// NETWORK 41
//   axisdata[4].Axis_Inbb: A-0-0021.13 -RD- Axis is ready for power to the amplifier (bb)
//   FP_C_0_0051: Operating hour counter
//   drive4: Real axis "Drive4" with axis number 4
//   r_operation_hour: FP_C_0_0051,Operation hour counter
fb_read_operation_hour(
    Enable := axisdata[4].Axis_Inbb,
    ParameterNumber := FP_C_0_0051,
    Axis := drive4,
    Value => r_operation_hour); // MB_ReadParameter

// NETWORK 42
//   axisdata[1].Axis_Inbb: A-0-0021.13 -RD- Axis is ready for power to the amplifier (bb)
//   FP_s_0_0189: Following distance
//   drive1: Real axis "Drive1" with axis number 1
//   r_following_11: FP_s_0_0189,following error
fb_read_s189_1(
    Enable := axisdata[1].Axis_Inbb,
    ParameterNumber := FP_s_0_0189,
    Axis := drive1,
    Value => r_following_11); // MB_ReadRealParameter

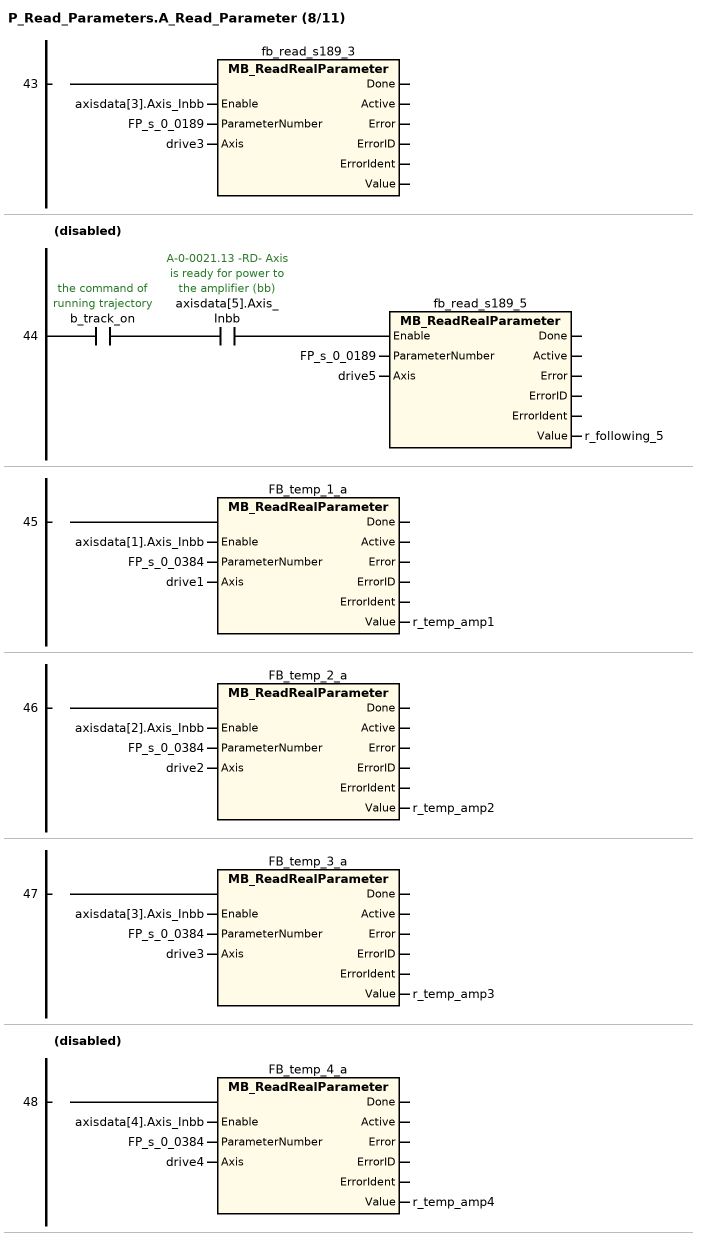
// NETWORK 43
//   axisdata[3].Axis_Inbb: A-0-0021.13 -RD- Axis is ready for power to the amplifier (bb)
//   FP_s_0_0189: Following distance
//   drive3: Real axis "Drive3" with axis number 3
fb_read_s189_3(Enable := axisdata[3].Axis_Inbb, ParameterNumber := FP_s_0_0189, Axis := drive3); // MB_ReadRealParameter

// NETWORK 44 (disabled)
//   b_track_on: the command of running trajectory
//   axisdata[5].Axis_Inbb: A-0-0021.13 -RD- Axis is ready for power to the amplifier (bb)
//   FP_s_0_0189: Following distance
//   drive5: Real axis "Drive5" with axis number 5
// fb_read_s189_5(
//     Enable := b_track_on AND axisdata[5].Axis_Inbb,
//     ParameterNumber := FP_s_0_0189,
//     Axis := drive5,
//     Value => r_following_5); // MB_ReadRealParameter

// NETWORK 45
//   axisdata[1].Axis_Inbb: A-0-0021.13 -RD- Axis is ready for power to the amplifier (bb)
//   FP_s_0_0384: Amplifier temperature
//   drive1: Real axis "Drive1" with axis number 1
//   r_temp_amp1: FP_S_0_0384,Amplifier temperature
FB_temp_1_a(
    Enable := axisdata[1].Axis_Inbb,
    ParameterNumber := FP_s_0_0384,
    Axis := drive1,
    Value => r_temp_amp1); // MB_ReadRealParameter

// NETWORK 46
//   axisdata[2].Axis_Inbb: A-0-0021.13 -RD- Axis is ready for power to the amplifier (bb)
//   FP_s_0_0384: Amplifier temperature
//   drive2: Real axis "Drive2" with axis number 2
FB_temp_2_a(
    Enable := axisdata[2].Axis_Inbb,
    ParameterNumber := FP_s_0_0384,
    Axis := drive2,
    Value => r_temp_amp2); // MB_ReadRealParameter

// NETWORK 47
//   axisdata[3].Axis_Inbb: A-0-0021.13 -RD- Axis is ready for power to the amplifier (bb)
//   FP_s_0_0384: Amplifier temperature
//   drive3: Real axis "Drive3" with axis number 3
FB_temp_3_a(
    Enable := axisdata[3].Axis_Inbb,
    ParameterNumber := FP_s_0_0384,
    Axis := drive3,
    Value => r_temp_amp3); // MB_ReadRealParameter

// NETWORK 48 (disabled)
//   axisdata[4].Axis_Inbb: A-0-0021.13 -RD- Axis is ready for power to the amplifier (bb)
//   FP_s_0_0384: Amplifier temperature
//   drive4: Real axis "Drive4" with axis number 4
// FB_temp_4_a(
//     Enable := axisdata[4].Axis_Inbb,
//     ParameterNumber := FP_s_0_0384,
//     Axis := drive4,
//     Value => r_temp_amp4); // MB_ReadRealParameter

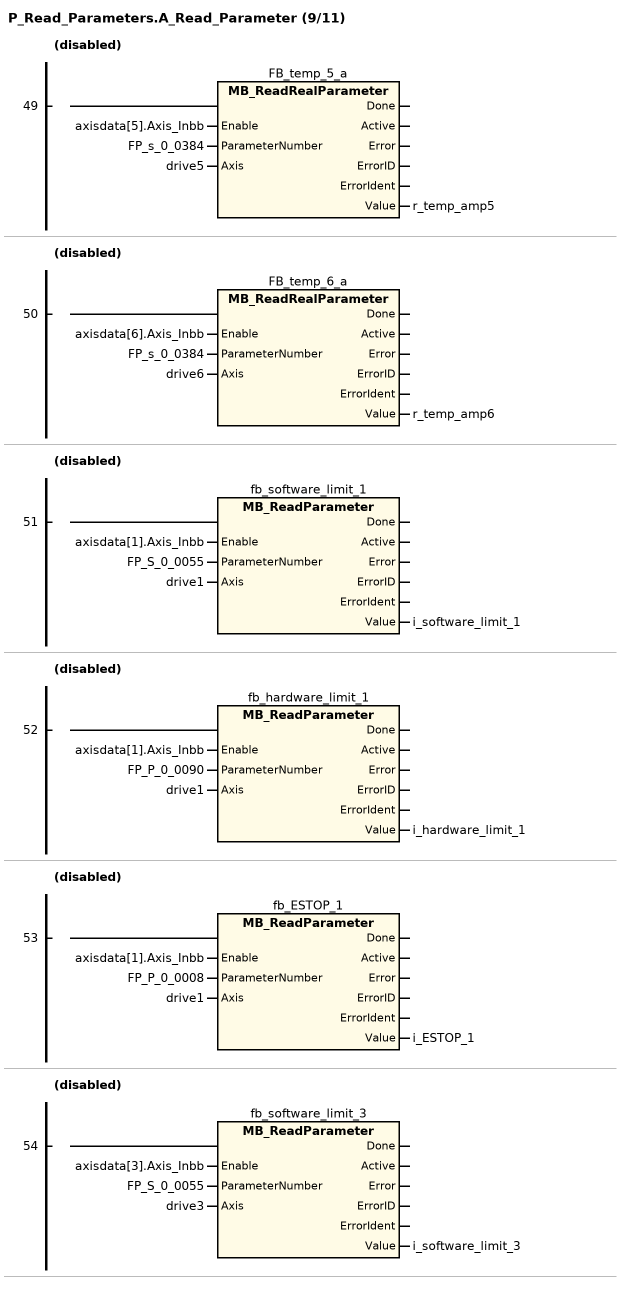
// NETWORK 49 (disabled)
//   axisdata[5].Axis_Inbb: A-0-0021.13 -RD- Axis is ready for power to the amplifier (bb)
//   FP_s_0_0384: Amplifier temperature
//   drive5: Real axis "Drive5" with axis number 5
// FB_temp_5_a(
//     Enable := axisdata[5].Axis_Inbb,
//     ParameterNumber := FP_s_0_0384,
//     Axis := drive5,
//     Value => r_temp_amp5); // MB_ReadRealParameter

// NETWORK 50 (disabled)
//   axisdata[6].Axis_Inbb: A-0-0021.13 -RD- Axis is ready for power to the amplifier (bb)
//   FP_s_0_0384: Amplifier temperature
//   drive6: Real axis "Drive6" with axis number 6
// FB_temp_6_a(
//     Enable := axisdata[6].Axis_Inbb,
//     ParameterNumber := FP_s_0_0384,
//     Axis := drive6,
//     Value => r_temp_amp6); // MB_ReadRealParameter

// NETWORK 51 (disabled)
//   fb_software_limit_1: test for limit check
//   axisdata[1].Axis_Inbb: A-0-0021.13 -RD- Axis is ready for power to the amplifier (bb)
//   FP_S_0_0055: Position polarities
//   drive1: Real axis "Drive1" with axis number 1
// fb_software_limit_1(
//     Enable := axisdata[1].Axis_Inbb,
//     ParameterNumber := FP_S_0_0055,
//     Axis := drive1,
//     Value => i_software_limit_1); // MB_ReadParameter

// NETWORK 52 (disabled)
//   axisdata[1].Axis_Inbb: A-0-0021.13 -RD- Axis is ready for power to the amplifier (bb)
//   FP_P_0_0090: Travel range limit parameter
//   drive1: Real axis "Drive1" with axis number 1
// fb_hardware_limit_1(
//     Enable := axisdata[1].Axis_Inbb,
//     ParameterNumber := FP_P_0_0090,
//     Axis := drive1,
//     Value => i_hardware_limit_1); // MB_ReadParameter

// NETWORK 53 (disabled)
//   axisdata[1].Axis_Inbb: A-0-0021.13 -RD- Axis is ready for power to the amplifier (bb)
//   FP_P_0_0008: Activation E-Stop function
//   drive1: Real axis "Drive1" with axis number 1
// fb_ESTOP_1(
//     Enable := axisdata[1].Axis_Inbb,
//     ParameterNumber := FP_P_0_0008,
//     Axis := drive1,
//     Value => i_ESTOP_1); // MB_ReadParameter

// NETWORK 54 (disabled)
//   axisdata[3].Axis_Inbb: A-0-0021.13 -RD- Axis is ready for power to the amplifier (bb)
//   FP_S_0_0055: Position polarities
//   drive3: Real axis "Drive3" with axis number 3
// fb_software_limit_3(
//     Enable := axisdata[3].Axis_Inbb,
//     ParameterNumber := FP_S_0_0055,
//     Axis := drive3,
//     Value => i_software_limit_3); // MB_ReadParameter

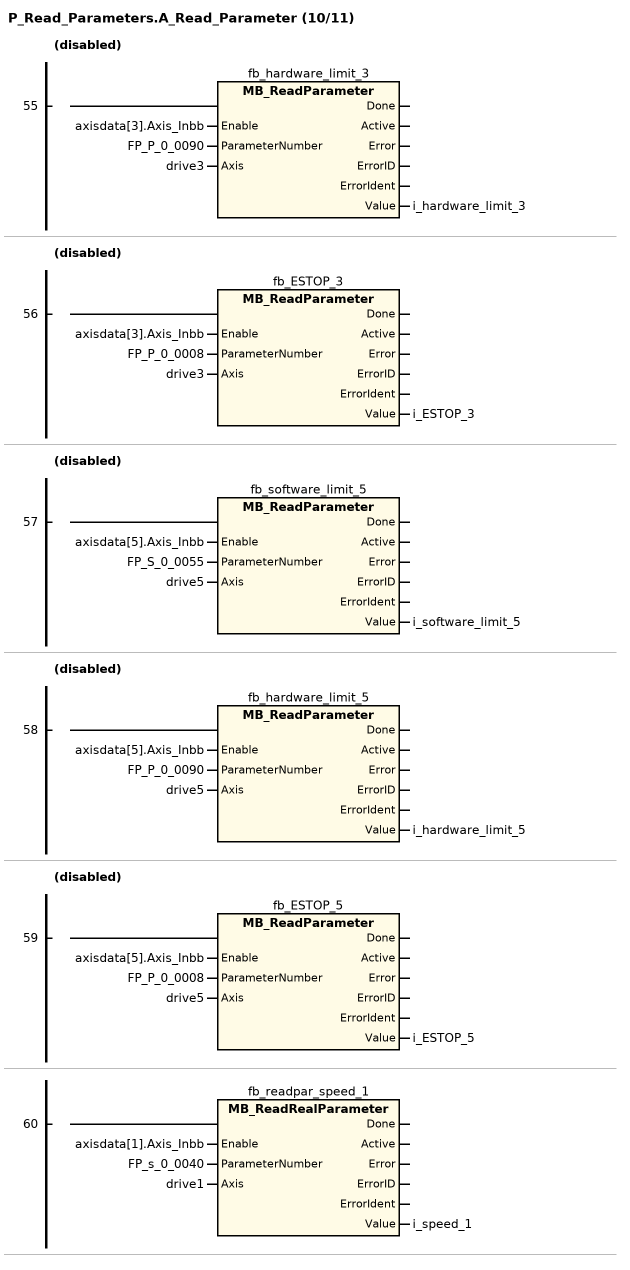
// NETWORK 55 (disabled)
//   axisdata[3].Axis_Inbb: A-0-0021.13 -RD- Axis is ready for power to the amplifier (bb)
//   FP_P_0_0090: Travel range limit parameter
//   drive3: Real axis "Drive3" with axis number 3
// fb_hardware_limit_3(
//     Enable := axisdata[3].Axis_Inbb,
//     ParameterNumber := FP_P_0_0090,
//     Axis := drive3,
//     Value => i_hardware_limit_3); // MB_ReadParameter

// NETWORK 56 (disabled)
//   axisdata[3].Axis_Inbb: A-0-0021.13 -RD- Axis is ready for power to the amplifier (bb)
//   FP_P_0_0008: Activation E-Stop function
//   drive3: Real axis "Drive3" with axis number 3
// fb_ESTOP_3(
//     Enable := axisdata[3].Axis_Inbb,
//     ParameterNumber := FP_P_0_0008,
//     Axis := drive3,
//     Value => i_ESTOP_3); // MB_ReadParameter

// NETWORK 57 (disabled)
//   axisdata[5].Axis_Inbb: A-0-0021.13 -RD- Axis is ready for power to the amplifier (bb)
//   FP_S_0_0055: Position polarities
//   drive5: Real axis "Drive5" with axis number 5
// fb_software_limit_5(
//     Enable := axisdata[5].Axis_Inbb,
//     ParameterNumber := FP_S_0_0055,
//     Axis := drive5,
//     Value => i_software_limit_5); // MB_ReadParameter

// NETWORK 58 (disabled)
//   axisdata[5].Axis_Inbb: A-0-0021.13 -RD- Axis is ready for power to the amplifier (bb)
//   FP_P_0_0090: Travel range limit parameter
//   drive5: Real axis "Drive5" with axis number 5
// fb_hardware_limit_5(
//     Enable := axisdata[5].Axis_Inbb,
//     ParameterNumber := FP_P_0_0090,
//     Axis := drive5,
//     Value => i_hardware_limit_5); // MB_ReadParameter

// NETWORK 59 (disabled)
//   axisdata[5].Axis_Inbb: A-0-0021.13 -RD- Axis is ready for power to the amplifier (bb)
//   FP_P_0_0008: Activation E-Stop function
//   drive5: Real axis "Drive5" with axis number 5
// fb_ESTOP_5(
//     Enable := axisdata[5].Axis_Inbb,
//     ParameterNumber := FP_P_0_0008,
//     Axis := drive5,
//     Value => i_ESTOP_5); // MB_ReadParameter

// NETWORK 60
//   axisdata[1].Axis_Inbb: A-0-0021.13 -RD- Axis is ready for power to the amplifier (bb)
//   FP_s_0_0040: Velocity feedback value
//   drive1: Real axis "Drive1" with axis number 1
//   i_speed_1: the velocity feedback value of motor1
fb_readpar_speed_1(
    Enable := axisdata[1].Axis_Inbb,
    ParameterNumber := FP_s_0_0040,
    Axis := drive1,
    Value => i_speed_1); // MB_ReadRealParameter

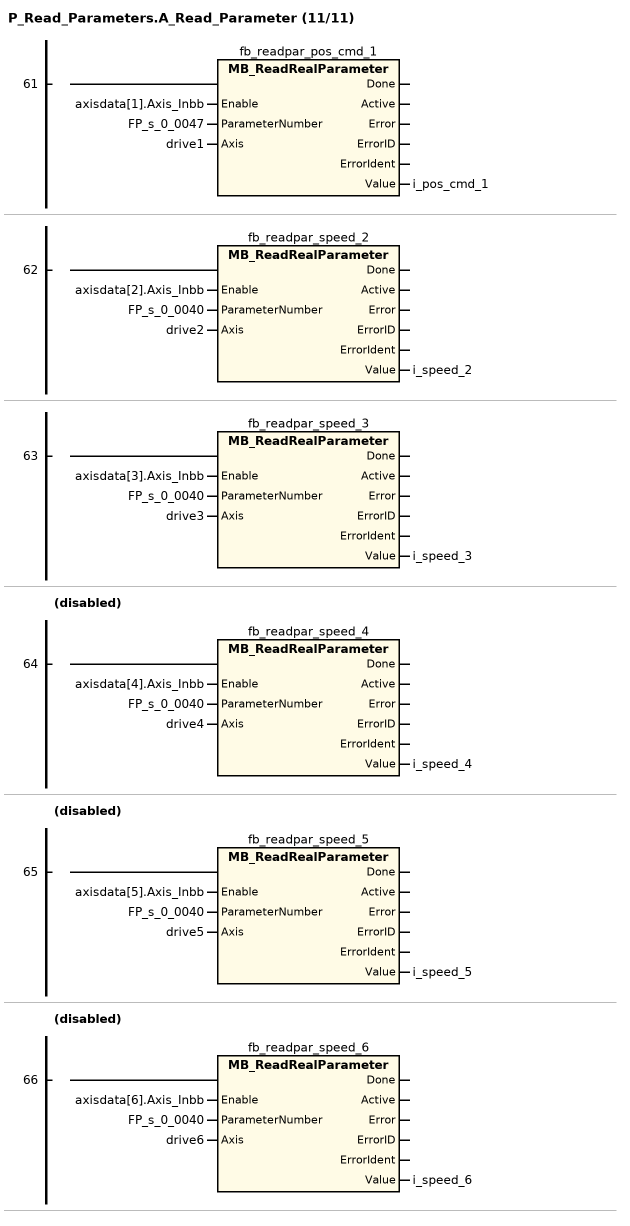
// NETWORK 61
//   axisdata[1].Axis_Inbb: A-0-0021.13 -RD- Axis is ready for power to the amplifier (bb)
//   FP_s_0_0047: Velocity feedback value
//   drive1: Real axis "Drive1" with axis number 1
//   i_pos_cmd_1: the velocity feedback value of motor1
fb_readpar_pos_cmd_1(
    Enable := axisdata[1].Axis_Inbb,
    ParameterNumber := FP_s_0_0047,
    Axis := drive1,
    Value => i_pos_cmd_1); // MB_ReadRealParameter

// NETWORK 62
//   axisdata[2].Axis_Inbb: A-0-0021.13 -RD- Axis is ready for power to the amplifier (bb)
//   FP_s_0_0040: Velocity feedback value
//   drive2: Real axis "Drive2" with axis number 2
//   i_speed_2: the velocity feedback value of motor1
fb_readpar_speed_2(
    Enable := axisdata[2].Axis_Inbb,
    ParameterNumber := FP_s_0_0040,
    Axis := drive2,
    Value => i_speed_2); // MB_ReadRealParameter

// NETWORK 63
//   axisdata[3].Axis_Inbb: A-0-0021.13 -RD- Axis is ready for power to the amplifier (bb)
//   FP_s_0_0040: Velocity feedback value
//   drive3: Real axis "Drive3" with axis number 3
//   i_speed_3: the velocity feedback value of motor3
fb_readpar_speed_3(
    Enable := axisdata[3].Axis_Inbb,
    ParameterNumber := FP_s_0_0040,
    Axis := drive3,
    Value => i_speed_3); // MB_ReadRealParameter

// NETWORK 64 (disabled)
//   axisdata[4].Axis_Inbb: A-0-0021.13 -RD- Axis is ready for power to the amplifier (bb)
//   FP_s_0_0040: Velocity feedback value
//   drive4: Real axis "Drive4" with axis number 4
//   i_speed_4: the velocity feedback value of motor1
// fb_readpar_speed_4(
//     Enable := axisdata[4].Axis_Inbb,
//     ParameterNumber := FP_s_0_0040,
//     Axis := drive4,
//     Value => i_speed_4); // MB_ReadRealParameter

// NETWORK 65 (disabled)
//   axisdata[5].Axis_Inbb: A-0-0021.13 -RD- Axis is ready for power to the amplifier (bb)
//   FP_s_0_0040: Velocity feedback value
//   drive5: Real axis "Drive5" with axis number 5
//   i_speed_5: the velocity feedback value of motor5
// fb_readpar_speed_5(
//     Enable := axisdata[5].Axis_Inbb,
//     ParameterNumber := FP_s_0_0040,
//     Axis := drive5,
//     Value => i_speed_5); // MB_ReadRealParameter

// NETWORK 66 (disabled)
//   axisdata[6].Axis_Inbb: A-0-0021.13 -RD- Axis is ready for power to the amplifier (bb)
//   FP_s_0_0040: Velocity feedback value
//   drive6: Real axis "Drive6" with axis number 6
//   i_speed_6: the velocity feedback value of motor1
// fb_readpar_speed_6(
//     Enable := axisdata[6].Axis_Inbb,
//     ParameterNumber := FP_s_0_0040,
//     Axis := drive6,
//     Value => i_speed_6); // MB_ReadRealParameter
END_ACTION

END_PROGRAM

// IndraMotionMlc1/Application/POUs/Motion/P_interpolator
(*This program is built for running trajectory,and the trajectory runs by the rule y=ax^2+bx+c.
In this PROGRAM,there are two kinds OF FUNCTION blocks,ML_WriteCyclicPosition AND ML_OpenCyclicPositionChannel.
They are used for give the position command value to the virtual axis.*)
PROGRAM P_interpolator
VAR
(*azimuth,elevation and FeedIndexer position at i_start point *)
	p1_az: LREAL;
	p1_el: LREAL;
	p1_FI: LREAL;
(*azimuth,elevation and FeedIndexer position at i_start+1 point*)
	p2_az: LREAL;
	p2_el: LREAL;
	p2_FI: LREAL;
(*azimuth,elevation and FeedIndexer position at i_start+2 point*)
	p3_az: LREAL;
	p3_el: LREAL;
	p3_FI: LREAL;
(*the facters of the formula y=ax^2+bx+c*)
	a_az: LREAL;
	b_az: LREAL;
	a_el: LREAL;
	b_el: LREAL;
	a_FI: LREAL;
	b_FI: LREAL;
	t: LREAL;
	t1: LREAL;(*the time at i_start point*)
	t2: LREAL;(*the time at i_start+1 point*)
	t3: LREAL;(*the time at i_start+2 point*)
	
(*<<<<<<<<<<<<<<<<<<<<<<<<Write a Position value to azimuth,elevation and FeedIndexer virtual axis>>>>>>>>>>>>>>>>>>*)
	fb_write_positon_az: ML_WriteCyclicPosition;
	fb_write_positon_el: ML_WriteCyclicPosition;
	fb_write_positon_FI: ML_WriteCyclicPosition;

(*Open Cyclic Position Channel for azimuth,elevation and FeedIndexer.
Only if the cyclic position target value channel is open, 
the position command will become effective in the next cycle on the axis.*)
	fb_open_channel_az: ML_OpenCyclicPositionChannel;
	fb_open_channel_el: ML_OpenCyclicPositionChannel;
	fb_open_channel_FI: ML_OpenCyclicPositionChannel;

(*<<<<<<<<<<<<<definition for rtrig>>>>>>>>>>>>>>*)
	rtrig_track_on: R_TRIG;
	rtrig_write_position: R_TRIG;
	rtrig_reset_open_channel: R_TRIG;
	rtrig_reset_goto_track: R_TRIG;
	r_rtrig_start_stop:R_TRIG;
	ton_track_on:TON;
	b_signal_for_open: BOOL;
(*<<<<<<<<<<<<<<<<<<<<<<<the current position>>>>>>>>>>>>>>>>>>>*)
	r_last_position_az: LREAL;
	r_last_position_el: LREAL;
	r_last_position_FI: LREAL;
(*<<<<<<<<<<<<<<<<<<<<<<<<<<the current speed>>>>>>>>>>>>>>>>>>>>*)
	r_vel_last_az: LREAL;
	r_vel_last_el: LREAL;
	r_vel_last_FI: LREAL;
(*the distance and time between the current point and the first point*)
	r_start_distance_az: LREAL;
	r_start_distance_el: LREAL;
	r_start_distance_FI: LREAL;
	r_time_distance: LREAL;
(*the current velocity *)
	r_vel_start_az: LREAL;
	r_vel_start_el: LREAL;
	r_vel_start_FI: LREAL;
(*the transition for the azimuth position,r_write_position_az.*)
	r_calc_pos_az:LREAL;
	V0_el: LREAL;
	V0_az: LREAL;
	V0_FI: LREAL;
	i_point_caught: INT:=1;
	V_start_az: LREAL;
	V_start_el: LREAL;
	V_start_FI: LREAL;
	i_caught_MJD1:LREAL;
	i_caught_MJD2:LREAL;
	i_caught_TAIoffset1:LREAL;
	i_caught_TAIoffset2:LREAL;
	b_test:BOOL;
	
	i_start_first:INT;
	i_end_first:INT;
	
	test_1:INT;
	test_2:INT;
	
	r_start_az:LREAL;
	r_caught_az:LREAL;
	
	ton_pause_on:TON;
	rtrig_pause_on:R_TRIG;
	r_abs_az_speed:LREAL; // units deg/sec
	r_abs_el_speed:LREAL; // units deg/sec
	test_enable_el: BOOL;
	b_start_to_compensate: BOOL;
	p_covert_velocity:LREAL;
	r_following_test: LREAL;
	r_following_31: LREAL;
	r_following_333: LREAL;
	p_covert_velocity_el: LREAL;	
	(**********offset************)
	r_az_offset_Vmax:LREAL:=2.0;
	r_el_offset_Vmax:LREAL:=0.85;
	r_az_offset_acc:LREAL:=1.0;
	r_el_offset_acc:LREAL:=0.25;
	r_az_offset_dec:LREAL:=0.5;
	r_el_offset_dec:LREAL:=0.25;
	r_old_offset_az:LREAL;
	r_old_offset_el:LREAL;
	r_new_offset_az:LREAL;
	r_new_offset_el:LREAL;

	r_test_offset_az_abs:LREAL;
	r_test_offset_el_abs:LREAL;
	i_test_offset_count:DINT:=0;
	r_offset_t1_acc:LREAL;
	r_offset_t2_v:LREAL;
	r_offset_t3_dec:LREAL;
	l_offset_t1_acc:LREAL;
	l_offset_t2_v:LREAL;
	l_offset_t3_dec:LREAL;
	r_offset_t1_acc_el:LREAL;
	r_offset_t2_v_el:LREAL;
	r_offset_t3_dec_el:LREAL;
	l_offset_t1_acc_el:LREAL;
	l_offset_t2_v_el:LREAL;
	l_offset_t3_dec_el:LREAL;
	r_offset_t:LREAL:=0;
	test_t:LREAL;
	r_az_offset_abs:LREAL;
	
	Static_done: BOOL;
	r_write_position_az_s: LREAL;
	r_write_position_el_s: LREAL;
	s_mp: StaticPmParam;
	Az_rad: LREAL;
	El_rad: LREAL;
	ABphi_rad: LREAL;
	TE: INT;
	//r_write_position_az_out: LREAL;
	//r_write_position_el_out: LREAL;
	test1: BOOL;
	Test2: BOOL;
	test3: BOOL;
	test4: BOOL;
	test5: BOOL;
	test6: BOOL;
	test7: BOOL;
	test8: BOOL;
	test9: BOOL;
	rtrig_write_position_sim: R_TRIG;
	fb_move_sim_track_Az: MC_MoveAbsolute;
	b_sim_trk_az_done: BOOL;
	b_sim_trk_el_done: BOOL;
	rtrig_reset_sim: R_TRIG;
	rtrig_reset_sim_move: R_TRIG;
	fb_move_sim_track_El: MC_MoveAbsolute;
	b_sim_write_az: BOOL;
	b_sim_trk_az_active: BOOL;
	TON_0: TON;
	b_sim_trk_el_active: BOOL;
	b_sim_trk_az_active_not: BOOL;
	f_trig_sim: F_TRIG;
	R_TRIG_0: R_TRIG;
	F_TRIG_0: F_TRIG;
	F_TRIG_1: F_TRIG;
	TON_1: TON;
	IL_EnableInOpBase_0: IL_SIGNALGENERATORTYPE01;
	TP_0: TP;
	TP_1: TP;
	TP_2: TP;
	BLINK_0: BLINK;
	b_sim_trk_exec: BOOL;
END_VAR

(*IF test_enable_el THEN
arAxisCtrl_gb[Drive3.AxisNo].Admin._OpMode.en := Modeah;
ELSE
arAxisCtrl_gb[Drive3.AxisNo].Admin._OpMode.en := Modeab;
END_IF
*)
//axisdata[3].dwUserCmdDataA_q.REAL_;

//axisdata[3].dwUserActualDataA_i.REAL_;



//axisdata[3].dwUserCmdDataA_q.REAL_:=axisdata[3].dwUserActualDataA_i.REAL_;





(*<<<<<<<<<<<<<<<<<<<<<calculate the current point in the stack>>>>>>>>>>>>>>>>>>>>>>>*)
//WHILE lr_MJD_current >= track_table[F_I_number(i_start+1)].MJD DO
test1:=lr_TAIoffset_current >= track_table[F_I_number(i_start+1)].TAIoffset;
WHILE lr_TAIoffset_current >= track_table[F_I_number(i_start+1)].TAIoffset DO
	IF i_start= i_end THEN
		EXIT;
	ELSE
		i_start:=F_I_number(i_start+1);
	END_IF;
END_WHILE


(*<<<<<<<<<<<<<<<<<<calculate the number of the points left in the stack>>>>>>>>>>>>>>*)
IF i_start=i_end THEN
	i_num_stack_left:=0;
ELSE
	i_num_stack_left:= i_end-i_start+1;
	IF i_num_stack_left<=0 THEN
		i_num_stack_left:=i_num_stack_left+i_total;
	END_IF;
END_IF

(* I Don't know what this piece of code is meant to do commenting it out 8/8/2024
IF i_num_stack_left>10 AND b_remote_on_run AND b_track_on=FALSE THEN
	b_track_on:=TRUE;
END_IF; *)


r_abs_az_speed:=ABS(AxisData[1].rActualVelocity_i)*6;
p_covert_velocity:=(0.5773*r_abs_az_speed*r_abs_az_speed*r_abs_az_speed - 0.4526*r_abs_az_speed*r_abs_az_speed + 11.313*r_abs_az_speed + 4.523)*0.2535;
p_covert_velocity_el:=0.5773*r_vel_EL*r_vel_EL*r_vel_EL - 0.4526*r_vel_EL*r_vel_EL + 11.313*r_vel_EL + 4.523;
(*<<<<<<<<<<<<<<<<<<<<<<<<<<<<<<<<<<<<<<the definication of trigger and TON>>>>>>>>>>>>>>>>>>>>>>>>>>>>>>>>>>>>>>>>>>>>>>>*)
r_rtrig_start_stop(clk:=b_track_on);(*before tracking ,stop the motion*)
ton_track_on(IN:=b_track_on,PT:=T#200MS);(*by using 200ms,program can search about 60 points*)
rtrig_track_on(clk:=ton_track_on.Q);(*the trigger for the initializtion*)


ton_pause_on(IN:=b_Track_Pause,PT:=T#4000MS);(*by using 200ms,program can search about 60 points*)
rtrig_pause_on(clk:=ton_pause_on.Q);(*the trigger for the initializtion*)

IF rtrig_pause_on.Q THEN
	b_track_on:=FALSE;
END_IF


(*<<<<<<<<<<<<<<<<<<<<<<<<<<<<main program of track>>>>>>>>>>>>>>>>>>>>>>>>>>>>>*)
IF b_track_on=TRUE THEN
	
(*<<<<<<<<<<<<<<<<<<<<<<<<<<< Calculate the tracking error>>>>>>>>>>>>>>>>>>>>>>>>>>>>>*)
	
	//IF ABS(track_table[i_start].MJD-lr_mjd_current)*86400<0.001 THEN
	Test2:=ABS(track_table[i_start].TAIoffset-lr_TAIoffset_current)<0.001;
	IF ABS(track_table[i_start].TAIoffset-lr_TAIoffset_current)<0.001 THEN
		r_following_1:=(r_pos_az_v-track_table[i_start].Azimuth);
		IF  ABS(r_following_1)<0.5  THEN
		   r_following_1:=(r_pos_az_v-track_table[i_start].Azimuth)/p_covert_velocity;
		END_IF
		   r_following_3:=(r_pos_el_v-track_table[i_start].Elevation);
		IF ABS(r_following_3)>0.0001 AND ABS(r_following_3)<=0.003 THEN
			r_following_3:=(r_pos_el_v-track_table[i_start].Elevation)/1.5;
		END_IF
		IF ABS(r_following_3)>0.003 AND ABS(r_following_3)<=0.006 THEN
			r_following_3:=(r_pos_el_v-track_table[i_start].Elevation)/2;
		END_IF
		IF ABS(r_following_3)>0.006 AND ABS(r_following_3)<=0.02 THEN
			r_following_3:=(r_pos_el_v-track_table[i_start].Elevation)/4;
		END_IF
		r_following_radius_asec := LREAL_TO_REAL((SQRT(EXPT(r_following_1,2)+EXPT(r_following_3,2)))*3600);  // Following erroring terms of a radius. 
	END_IF
(*
	IF ABS(r_following_3)> ABS(r_track_error[2]) THEN	
		r_following_33:=r_track_error[2];
	ELSE
		r_following_33:=r_following_33;
	END_IF
		IF ABS(r_following_33)>0.01 THEN
			r_following_33:=r_following_33/10;
		END_IF
	IF ABS(r_vel_EL)<0.0001 THEN
		r_following_3:=r_following_33;
	ELSE
		r_following_3:=r_following_33/p_covert_velocity_el;
	END_IF	
*)	
(*<<<<<<<<<<<<when finish all the points or the power is down,then reset the track_on>>>>>>>>>>>>>>>>>>>*)
	IF i_start=i_end OR b_remote_on_run=FALSE THEN
		 b_track_on:=FALSE;
	END_IF
(*<<<<<<<<<<<<<<<<<<<<<<<<<<<<stop the motion before tracking>>>>>>>>>>>>>>>>>>>*)
	IF r_rtrig_start_stop.Q THEN
		b_SCC_STOP:=TRUE;
	END_IF
	IF rtrig_track_on.Q=TRUE THEN
(*<<<<<<<<<<<<<<<<<<<<<<<<<<<<<<find the first point which can be caught up>>>>>>>>>>>>>>>>>>>>>>>>>>>*)
		//WHILE ABS(track_table[i_start].Azimuth-r_pos_az_v)/((track_table[i_start].MJD-lr_mjd_current)*86400-0.05)>2.9 OR (track_table[i_start].MJD-lr_mjd_current)*86400-0.05<0 DO
		test3:=ABS(track_table[i_start].Azimuth-r_pos_az_v)/((track_table[i_start].TAIoffset-lr_TAIoffset_current)-0.05)>2.9 OR (track_table[i_start].TAIoffset-lr_TAIoffset_current)-0.05<0;
		WHILE ABS(track_table[i_start].Azimuth-r_pos_az_v)/((track_table[i_start].TAIoffset-lr_TAIoffset_current)-0.05)>2.9 OR (track_table[i_start].TAIoffset-lr_TAIoffset_current)-0.05<0 DO
		//WHILE ABS(entry_buffer1[i_start].Azimuth-r_pos_az_v)/((entry_buffer1[i_start].MJD-lr_mjd_current)*86400-0.05)>2.9 DO
			IF i_start=i_end-3 THEN
				EXIT;
			ELSE
				i_start:=F_I_number(i_start+1);
			END_IF
		END_WHILE
		
		//WHILE ABS(track_table[i_start].Elevation-r_pos_el)/((track_table[i_start].MJD-lr_mjd_current)*86400-0.05)>0.8 OR (track_table[i_start].MJD-lr_mjd_current)*86400-0.05<0 DO
		test4:=ABS(track_table[i_start].Elevation-r_pos_el)/((track_table[i_start].TAIoffset-lr_TAIoffset_current)-0.05)>0.8 OR (track_table[i_start].TAIoffset-lr_TAIoffset_current)-0.05<0;
		WHILE ABS(track_table[i_start].Elevation-r_pos_el)/((track_table[i_start].TAIoffset-lr_TAIoffset_current)-0.05)>0.8 OR (track_table[i_start].TAIoffset-lr_TAIoffset_current)-0.05<0 DO	
		//WHILE ABS(entry_buffer1[i_start].Elevation-r_pos_motor3)/((entry_buffer1[i_start].MJD-lr_mjd_current)*86400-0.05)>1000 DO
			IF i_start=i_end-3 THEN
				EXIT;
			ELSE
				i_start:=F_I_number(i_start+1);
			END_IF
		END_WHILE
(*		WHILE ABS(entry_buffer1[i_start].FeedIndexer-r_pos_FI_v)/((entry_buffer1[i_start].MJD-lr_mjd_current)*86400-0.05)>2 OR (entry_buffer1[i_start].MJD-lr_mjd_current)*86400-0.05<0 DO
			IF i_start=i_end-3 THEN
				EXIT;
			ELSE
				i_start:=F_I_number(i_start+1);
			END_IF
		END_WHILE
*)

//		arAxisCtrl_gb[Drive3.AxisNo].Admin._OpMode.en := ModeCyclicVelocity; 
		b_write_el_vel:=TRUE;
		i_point_caught:=i_start;
		//i_caught_MJD1:=track_table[i_point_caught].MJD;
		 i_caught_TAIoffset1:=track_table[i_point_caught].TAIoffset;
		//i_caught_MJD2:=lr_MJD_current;
		i_caught_TAIoffset2:=lr_TAIoffset_current;
		r_start_az:=r_pos_az_v;
		r_caught_az:=track_table[i_point_caught].Azimuth;
		
(*if the first point which can be caught up is the last one£¬reset track_on*)
		IF i_start=i_end-3 THEN
			b_track_on:=FALSE;
		ELSE
			//track_table[F_I_number(i_start-1)].MJD:=lr_MJD_current+0.0000008;(*(69ms)after gunner change p41 from 0 to 100ms*)
			track_table[F_I_number(i_start-1)].TAIoffset:=lr_TAIoffset_current+0.069;(*(69ms)after gunner change p41 from 0 to 100ms*)
			track_table[F_I_number(i_start-1)].Azimuth:=r_pos_az_v;
			track_table[F_I_number(i_start-1)].elevation:=r_pos_el;
(*			entry_buffer1[F_I_number(i_start-1)].FeedIndexer:=r_pos_FI_v;  *)
		i_start:=F_I_number(i_start-1);
		r_write_position_az:=track_table[i_start].Azimuth;
		r_write_position_el:=track_table[i_start].Elevation;
(*		r_write_position_FI:=entry_buffer1[i_start].FeedIndexer;   *)
		r_last_position_az:=r_write_position_az;
		r_last_position_el:=r_write_position_el;
(*		r_last_position_FI:=r_write_position_FI;   *)
		b_signal_for_open:=TRUE;
		END_IF

	END_IF
(*when the position is all nearby the start point,open the channel for writing position to all axis*)
test5:=b_signal_for_open AND (ABS(r_pos_az_v-track_table[i_start].Azimuth)<0.001) AND (ABS(r_pos_el-track_table[i_start].Elevation)<0.001);
	IF b_signal_for_open AND (ABS(r_pos_az_v-track_table[i_start].Azimuth)<0.001) AND (ABS(r_pos_el-track_table[i_start].Elevation)<0.001) THEN
		b_open_channel_az:=TRUE;
//		b_start_cyclicvel:=TRUE;
//		b_open_channel_el:=TRUE;
(*		b_open_channel_FI:=TRUE;*)
		b_signal_for_open:=FALSE;
	END_IF
(*defind the variables for calculating the cubic fuction*)
		//t:=lr_MJD_current;
		//t1:=track_table[i_start].MJD;
		//t2:=track_table[F_I_number(i_start+1)].MJD;
		//t3:=track_table[F_I_number(i_start+2)].MJD;
		t:=lr_TAIoffset_current;
		t1:=track_table[i_start].TAIoffset;
		t2:=track_table[F_I_number(i_start+1)].TAIoffset;
		t3:=track_table[F_I_number(i_start+2)].TAIoffset;
		p1_az:=track_table[i_start].Azimuth;
		p2_az:=track_table[F_I_number(i_start+1)].Azimuth;
		p3_az:=track_table[F_I_number(i_start+2)].Azimuth;
		
		r_test1:=p1_az;
		r_test2:=p2_az;
		r_test3:=p3_az;
		
		p1_el:=track_table[i_start].elevation;
		p2_el:=track_table[F_I_number(i_start+1)].elevation;
		p3_el:=track_table[F_I_number(i_start+2)].elevation;		
(*		p1_FI:=entry_buffer1[i_start].FeedIndexer;
		p2_FI:=entry_buffer1[F_I_number(i_start+1)].FeedIndexer;
		p3_FI:=entry_buffer1[F_I_number(i_start+2)].FeedIndexer;
*)		
		//i_start;
		test_1:=F_I_number(i_start+1);
		test_2:=F_I_number(i_start+2);
(*construct the first cubic section by 2 points and 2 velocity*)
(*	IF	lr_MJD_current<entry_buffer1[i_point_caught].MJD AND lr_MJD_current>entry_buffer1[F_I_number(i_point_caught-1)].MJD THEN  *)
	//IF	lr_MJD_current<i_caught_MJD1 AND lr_MJD_current>i_caught_MJD2 THEN
test6:=lr_TAIoffset_current<i_caught_TAIoffset1 AND lr_TAIoffset_current>i_caught_TAIoffset2;
 IF	lr_TAIoffset_current<i_caught_TAIoffset1 AND lr_TAIoffset_current>i_caught_TAIoffset2 THEN	
	
		IF b_track_on THEN
			V_start_az:=(p3_az-p2_az)/(t3-t2);
			V_start_el:=(p3_el-p2_el)/(t3-t2);
(*			V_start_FI:=(p3_FI-p2_FI)/(t3-t2);  *)
			v0_az:=V_start_az;
			v0_el:=V_start_el;
(*			v0_FI:=V_start_FI;   *)
			b_test:=TRUE;
			b_start_to_compensate:=TRUE;

			a_az:=V_start_az/(t2-t1)/(t2-t1)-2*(p2_az-p1_az)/(t2-t1)/(t2-t1)/(t2-t1);
			b_az:=3*(p2_az-p1_az)/(t2-t1)/(t2-t1)-V_start_az/(t2-t1);
			a_el:=V_start_el/(t2-t1)/(t2-t1)-2*(p2_el-p1_el)/(t2-t1)/(t2-t1)/(t2-t1);
			b_el:=3*(p2_el-p1_el)/(t2-t1)/(t2-t1)-V_start_el/(t2-t1);
(*			a_FI:=V_start_FI/(t2-t1)/(t2-t1)-2*(p2_FI-p1_FI)/(t2-t1)/(t2-t1)/(t2-t1);
			b_FI:=3*(p2_FI-p1_FI)/(t2-t1)/(t2-t1)-V_start_FI/(t2-t1);
*)
			r_write_position_az:=a_az*(t-t1)*(t-t1)*(t-t1)+b_az*(t-t1)*(t-t1)+p1_az;
			r_write_position_el:=a_el*(t-t1)*(t-t1)*(t-t1)+b_el*(t-t1)*(t-t1)+p1_el;
(*			r_write_position_FI:=a_FI*(t-t1)*(t-t1)*(t-t1)+b_FI*(t-t1)*(t-t1)+p1_FI;   *)
		END_IF
	ELSE
		IF i_num_stack_left>2 THEN
			IF b_track_on THEN
(*<<<<<<<<<<<<<<<<<<<<<<<<<<<<<calculate the a and b in the function y=ax^3+bx^2+cx+d>>>>>>>>>>>>>>>>>>>>>>*)
(*y=a*(x-x1)^3+b*(x-x1)^2+c(x-x1)+d,   c=v0,  d=y1*)
			a_az:=((p3_az-p1_az)/(t3-t1)/(t3-t1)-(p2_az-p1_az)/(t2-t1)/(t2-t1)-v0_az/(t3-t1)+v0_az/(t2-t1))/(t3-t2);
			b_az:=((p3_az-p1_az)*(t2-t1)/(t3-t1)/(t3-t1)-(p2_az-p1_az)*(t3-t1)/(t2-t1)/(t2-t1)-v0_az*(t2-t1)/(t3-t1)+v0_az*(t3-t1)/(t2-t1))/(t2-t3);
			a_el:=((p3_el-p1_el)/(t3-t1)/(t3-t1)-(p2_el-p1_el)/(t2-t1)/(t2-t1)-v0_el/(t3-t1)+v0_el/(t2-t1))/(t3-t2);
			b_el:=((p3_el-p1_el)*(t2-t1)/(t3-t1)/(t3-t1)-(p2_el-p1_el)*(t3-t1)/(t2-t1)/(t2-t1)-v0_el*(t2-t1)/(t3-t1)+v0_el*(t3-t1)/(t2-t1))/(t2-t3);
(*			a_FI:=((p3_FI-p1_FI)/(t3-t1)/(t3-t1)-(p2_FI-p1_FI)/(t2-t1)/(t2-t1)-v0_FI/(t3-t1)+v0_FI/(t2-t1))/(t3-t2);
			b_FI:=((p3_FI-p1_FI)*(t2-t1)/(t3-t1)/(t3-t1)-(p2_FI-p1_FI)*(t3-t1)/(t2-t1)/(t2-t1)-v0_FI*(t2-t1)/(t3-t1)+v0_FI*(t3-t1)/(t2-t1))/(t2-t3);
*)
b_test:=FALSE;
			//IF lr_MJD_current>=track_table[i_start].MJD AND lr_MJD_current<=track_table[F_I_number(i_start+1)].MJD THEN
			test7:=lr_TAIoffset_current>=track_table[i_start].TAIoffset AND lr_TAIoffset_current<=track_table[F_I_number(i_start+1)].TAIoffset;
			IF lr_TAIoffset_current>=track_table[i_start].TAIoffset AND lr_TAIoffset_current<=track_table[F_I_number(i_start+1)].TAIoffset THEN
			
				r_write_position_az:=a_az*(t-t1)*(t-t1)*(t-t1)+b_az*(t-t1)*(t-t1)+v0_az*(t-t1)+p1_az;
				r_write_position_el:=a_el*(t-t1)*(t-t1)*(t-t1)+b_el*(t-t1)*(t-t1)+v0_el*(t-t1)+p1_el;
				r_cyclic_velocity_test:=(p2_el-p1_el)/(t2-t1)/86400;
				//r_cyclic_velocity_test:=(p2_el-p1_el)/(t2-t1);
				r_cyclic_velocity:=V0_el/86400;
				// r_cyclic_velocity:=V0_el;
(*				r_write_position_FI:=a_FI*(t-t1)*(t-t1)*(t-t1)+b_FI*(t-t1)*(t-t1)+v0_FI*(t-t1)+p1_FI;   *)
			END_IF
(*calculate the velocity of the last point*)
			//IF (lr_MJD_current-track_table[F_I_number(i_start+1)].MJD)*86400>=-0.002 AND (lr_MJD_current-track_table[F_I_number(i_start+1)].MJD)*86400<0 THEN
			test8:=(lr_TAIoffset_current-track_table[F_I_number(i_start+1)].TAIoffset)>=-0.002 AND (lr_TAIoffset_current-track_table[F_I_number(i_start+1)].TAIoffset)<0;
			IF (lr_TAIoffset_current-track_table[F_I_number(i_start+1)].TAIoffset)>=-0.002 AND (lr_TAIoffset_current-track_table[F_I_number(i_start+1)].TAIoffset)<0 THEN
				V0_az:=3*a_az*(t2-t1)*(t2-t1)+2*b_az*(t2-t1)+v0_az;
				V0_el:=3*a_el*(t2-t1)*(t2-t1)+2*b_el*(t2-t1)+v0_el;
(*				V0_FI:=3*a_FI*(t2-t1)*(t2-t1)+2*b_FI*(t2-t1)+v0_FI;    *)
			END_IF
			END_IF
		ELSE
(*<<<<<<<<<<<<<<<<<<<<<<<<run the last two points>>>>>>>>>>>>>>>>>>>>>>>>>>*)
			IF b_track_on THEN 
				//IF lr_MJD_current>=track_table[i_start].MJD AND lr_MJD_current<=track_table[F_I_number(i_start+1)].MJD THEN
				test9:= lr_TAIoffset_current>=track_table[i_start].TAIoffset AND lr_TAIoffset_current<=track_table[F_I_number(i_start+1)].TAIoffset;
				IF lr_TAIoffset_current>=track_table[i_start].TAIoffset AND lr_TAIoffset_current<=track_table[F_I_number(i_start+1)].TAIoffset THEN
				r_write_position_az:=(p2_az-p1_az)*(t-t1)/(t2-t1)+p1_az;
				r_write_position_el:=(p2_el-p1_el)*(t-t1)/(t2-t1)+p1_el;
(*				r_write_position_FI:=((p2_FI-p1_FI)*(t-t1)/(t2-t1)+p1_FI);     *)
				END_IF
			END_IF
		END_IF
	END_IF

	
IF b_start_to_compensate THEN
//	r_offset_el:=r_compensation_value_motor;
	r_write_position_az:=r_write_position_az+r_test_offset_az;
	r_write_position_el:=r_write_position_el+r_test_offset_el;
//	r_write_position_el:=r_write_position_el+r_offset_el;
END_IF
	
(*<<<<<<<<<<<<<<<<<<<<<<<<<limit the trajectory speed >>>>>>>>>>>>>>>>>>>>>>>>>*)
(*Because the program runs every 2ms,so wo can limit the position by the rule ¦¤y<v*¦¤t.*)
(*Azimuth trajectory speed limit is 5.1¡ã/s*)


		IF r_write_position_az-r_last_position_az>0.0031 THEN
				r_write_position_az:=r_last_position_az+0.0031;
				b_track_overspeed_az:=1;
			ELSIF r_write_position_az-r_last_position_az<-0.0031 THEN
				r_write_position_az:=r_last_position_az-0.0031;
				b_track_overspeed_az:=1;
			ELSE
				b_track_overspeed_az:=0;
			END_IF
(*Elevation trajectory speed limit is 1.05¡ã/s*)
			IF r_write_position_el-r_last_position_el>0.00091 THEN
				r_write_position_el:=r_last_position_el+0.00091;
				b_track_overspeed_el:=1;
			ELSIF r_write_position_el-r_last_position_el<-0.00091 THEN
				r_write_position_el:=r_last_position_el-0.00091;
				b_track_overspeed_el:=1;
			ELSE
				b_track_overspeed_el:=0;
			END_IF
(*
(*FeedIndexer trajectory speed limit is 2.1¡ã/s*)
			IF r_write_position_FI-r_last_position_FI>0.0042 THEN
				r_write_position_FI:=r_last_position_FI+0.0042;
				b_track_overspeed_FI:=1;
			ELSIF r_write_position_FI-r_last_position_FI<-0.0042 THEN
				r_write_position_FI:=r_last_position_FI-0.0042;
				b_track_overspeed_FI:=1;
			ELSE
				b_track_overspeed_FI:=0;
			END_IF
*)
			
			
(*register the velocity and position for calculate the speed limit and acceleration limit*)
			r_last_position_az:=r_write_position_az;
			r_last_position_el:=r_write_position_el;
(*			r_last_position_FI:=r_write_position_FI;   *)
(*<<<<<<<<<<<<<<<<<<<<<<<<close the cyclic channel and reset the track error>>>>>>>>>>>>>>>>>>>>>>>>>>*)
ELSE
(*close the cyclic channel*)
	b_open_channel_az:=FALSE;
	b_open_channel_el:=FALSE;
	b_start_to_compensate:=FALSE;
	r_compensation_value_motor:=0;
(*	b_open_channel_FI:=FALSE;  *)
(*reset the following error and so on*)
    r_write_position_el:= axisdata[8].rActualPosition_i;
	r_write_position_az:=  axisdata[7].rActualPosition_i;
	r_track_error[1]:=0;
	r_track_error[2]:=0;
	r_track_error[3]:=0;
	V0_az:=0;
	V0_el:=0;
	V_start_az:=0;
	V_start_el:=0;
	IF NOT(b_SCC_goto) AND NOT(b_track_on) THEN 
		r_following_1:=0.00;
		r_following_3:=0.00;
	END_IF
END_IF

 IF  b_test_offset_start THEN
	 	r_offset_t:=r_offset_t+0.001;
		test_t:=r_offset_t-r_offset_t1_acc-r_offset_t2_v;
 		(*****************AZ offset**********)
		r_az_offset_abs:=ABS(r_offset_az);
		r_offset_t1_acc:=r_az_offset_Vmax/r_az_offset_acc;
	 	r_offset_t3_dec:=r_az_offset_Vmax/r_az_offset_dec;
	 	l_offset_t1_acc:=0.5*r_az_offset_acc*r_offset_t1_acc*r_offset_t1_acc;
	 	l_offset_t3_dec:=0.5*r_az_offset_dec*r_offset_t3_dec*r_offset_t3_dec;
 		r_offset_t2_v:=(r_az_offset_abs-l_offset_t1_acc-l_offset_t3_dec)/r_az_offset_Vmax;
		l_offset_t2_v:=r_az_offset_Vmax*r_offset_t2_v;

			IF r_offset_t <=r_offset_t1_acc THEN
				r_test_offset_az_abs:=0.5*r_az_offset_acc*r_offset_t*r_offset_t;
			ELSIF r_offset_t1_acc<r_offset_t AND r_offset_t<(r_offset_t1_acc+r_offset_t2_v) THEN 
				r_test_offset_az_abs:=r_test_offset_az_abs+0.001*r_az_offset_Vmax;
			ELSIF (r_offset_t1_acc+r_offset_t2_v)<=r_offset_t AND r_offset_t<(r_offset_t1_acc+r_offset_t2_v+r_offset_t3_dec) THEN
				r_test_offset_az_abs:=l_offset_t1_acc+l_offset_t2_v+(r_offset_t-r_offset_t1_acc-r_offset_t2_v)*r_az_offset_Vmax-0.5*r_az_offset_dec*(r_offset_t-r_offset_t1_acc-r_offset_t2_v)*(r_offset_t-r_offset_t1_acc-r_offset_t2_v);
			ELSE 
				r_test_offset_az_abs:=r_az_offset_abs;
			END_IF

		IF r_test_offset_az_abs>=r_az_offset_abs THEN
			r_test_offset_az_abs:=r_az_offset_abs;
		END_IF
		IF r_offset_az<0 THEN
			r_test_offset_az:=-r_test_offset_az_abs;
		ELSE 
			r_test_offset_az:=r_test_offset_az_abs;
		END_IF
		r_test_offset_az:=r_offset_az_old+r_test_offset_az;
		
		
			(*****************EL offset**********)
		r_el_offset_abs:=ABS(r_offset_el);
		r_offset_t1_acc_el:=r_el_offset_Vmax/r_el_offset_acc;
	 	r_offset_t3_dec_el:=r_el_offset_Vmax/r_el_offset_dec;
	 	l_offset_t1_acc_el:=0.5*r_el_offset_acc*r_offset_t1_acc_el*r_offset_t1_acc_el;
	 	l_offset_t3_dec_el:=0.5*r_el_offset_dec*r_offset_t3_dec_el*r_offset_t3_dec_el;
 		r_offset_t2_v_el:=(r_el_offset_abs-l_offset_t1_acc_el-l_offset_t3_dec_el)/r_el_offset_Vmax;
		l_offset_t2_v_el:=r_el_offset_Vmax*r_offset_t2_v_el;

			IF r_offset_t <=r_offset_t1_acc_el THEN
				r_test_offset_el_abs:=0.5*r_el_offset_acc*r_offset_t*r_offset_t;
			ELSIF r_offset_t1_acc_el<r_offset_t AND r_offset_t<(r_offset_t1_acc_el+r_offset_t2_v_el) THEN 
				r_test_offset_el_abs:=r_test_offset_el_abs+0.001*r_el_offset_Vmax;
			ELSIF (r_offset_t1_acc_el+r_offset_t2_v_el)<=r_offset_t AND r_offset_t<(r_offset_t1_acc_el+r_offset_t2_v_el+r_offset_t3_dec_el) THEN
				r_test_offset_el_abs:=l_offset_t1_acc_el+l_offset_t2_v_el+(r_offset_t-r_offset_t1_acc_el-r_offset_t2_v_el)*r_el_offset_Vmax-0.5*r_el_offset_dec*(r_offset_t-r_offset_t1_acc_el-r_offset_t2_v_el)*(r_offset_t-r_offset_t1_acc_el-r_offset_t2_v_el);
			ELSE 
				r_test_offset_el_abs:=r_el_offset_abs;
			END_IF

		IF r_test_offset_el_abs>=r_el_offset_abs THEN
			r_test_offset_el_abs:=r_el_offset_abs;
		END_IF
		IF r_offset_el<0 THEN
			r_test_offset_el:=-r_test_offset_el_abs;
		ELSE 
			r_test_offset_el:=r_test_offset_el_abs;
		END_IF
		r_test_offset_el:=r_offset_el_old+r_test_offset_el;
    IF 	r_test_offset_el_abs=r_el_offset_abs AND r_test_offset_az_abs=r_az_offset_abs THEN 	
		b_test_offset_start:=FALSE;
		b_offset_running:=FALSE;
	END_IF
				
ELSE
	i_test_offset_count:=0;
	r_offset_t:=0;
	r_offset_az_old:=r_test_offset_az;
	r_offset_el_old:=r_test_offset_el;
END_IF


P_Track_cubic.A_StaticPM();
P_Track_cubic.A_AmbTempPM();
P_Track_cubic.A_DynamicPM();


Tracking.Status.p_desired_El:=r_write_position_el-Tracking.Status.act_statOffset_value_El/gc_lr_arcsec2deg;
Tracking.Status.p_desired_Az:=r_write_position_az-(Tracking.Status.act_statOffset_value_Xel/gc_lr_arcsec2deg)/COS(ML_degtorad(r_write_position_el));

IF b_track_on THEN 
r_write_position_az_out:=r_write_position_az-Pointing.Status.StaticPmCorrVal_Az/gc_lr_arcsec2deg-Pointing.Status.TiltCorrVal_Az/gc_lr_arcsec2deg-Pointing.Status.AmbTempCorrVal_Az/gc_lr_arcsec2deg;
r_write_position_el_out:=r_write_position_el-Pointing.Status.StaticPmCorrVal_El/gc_lr_arcsec2deg-Pointing.Status.TiltCorrVal_El/gc_lr_arcsec2deg-Pointing.Status.AmbTempCorrVal_El/gc_lr_arcsec2deg;
END_IF

IF gc_b_sim_on THEN 
	P_Track_cubic.A_Sim_track_function_blocks();
ELSE	
	P_Track_cubic.A_track_fuction_blocks();
END_IF

ACTION A_track_fuction_blocks:
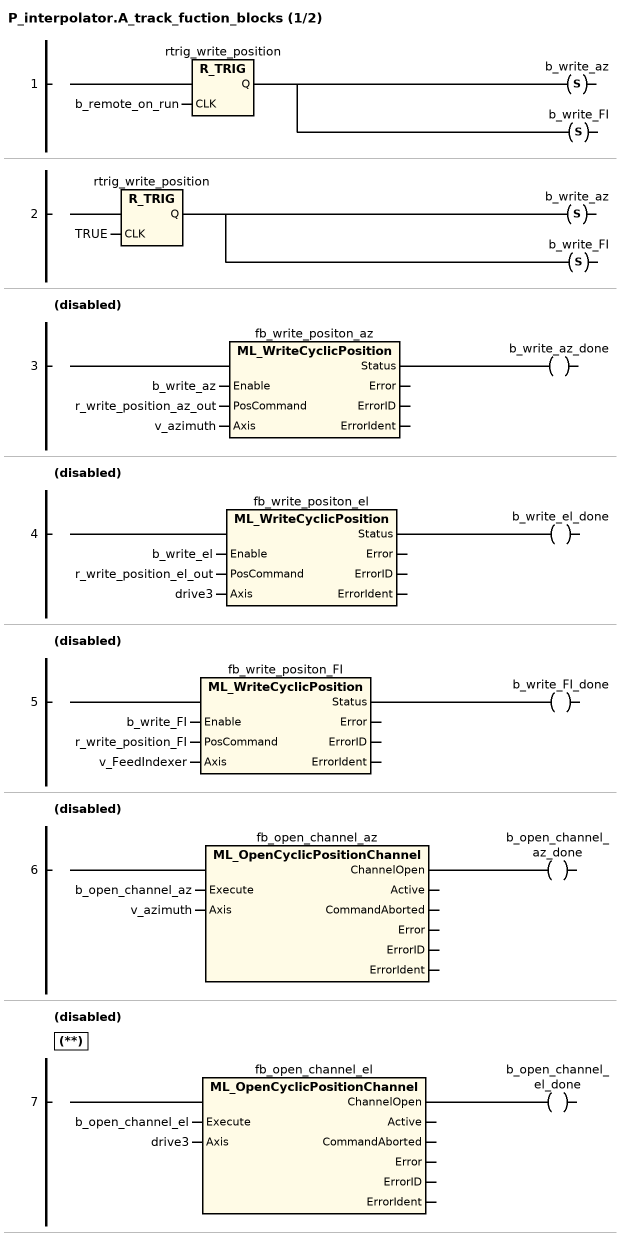
// NETWORK 1
rtrig_write_position(CLK := b_remote_on_run); // R_TRIG
b_write_az S= rtrig_write_position.Q;
b_write_FI S= rtrig_write_position.Q;

// NETWORK 2
rtrig_write_position(CLK := TRUE); // R_TRIG
b_write_az S= rtrig_write_position.Q;
b_write_FI S= rtrig_write_position.Q;

// NETWORK 3 (disabled)
// fb_write_positon_az(Enable := b_write_az, PosCommand := r_write_position_az_out, Axis := v_azimuth); // ML_WriteCyclicPosition
// b_write_az_done := fb_write_positon_az.Status;

// NETWORK 4 (disabled)
// fb_write_positon_el(Enable := b_write_el, PosCommand := r_write_position_el_out, Axis := drive3); // ML_WriteCyclicPosition
// b_write_el_done := fb_write_positon_el.Status;

// NETWORK 5 (disabled)
// fb_write_positon_FI(Enable := b_write_FI, PosCommand := r_write_position_FI, Axis := v_FeedIndexer); // ML_WriteCyclicPosition
// b_write_FI_done := fb_write_positon_FI.Status;

// NETWORK 6 (disabled)
// fb_open_channel_az(Execute := b_open_channel_az, Axis := v_azimuth); // ML_OpenCyclicPositionChannel
// b_open_channel_az_done := fb_open_channel_az.ChannelOpen;

// NETWORK 7 (disabled)
// label: (**)
// fb_open_channel_el(Execute := b_open_channel_el, Axis := drive3); // ML_OpenCyclicPositionChannel
// b_open_channel_el_done := fb_open_channel_el.ChannelOpen;

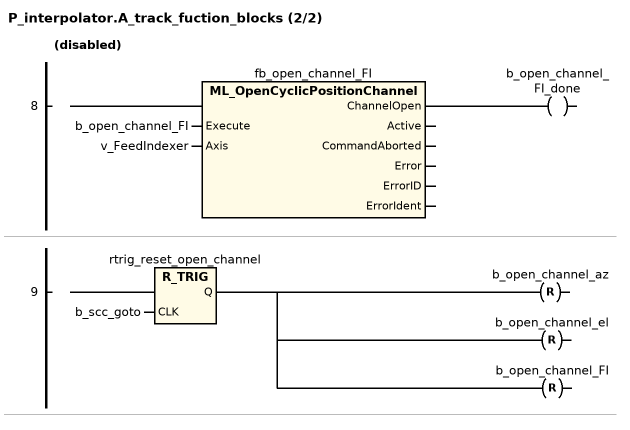
// NETWORK 8 (disabled)
// fb_open_channel_FI(Execute := b_open_channel_FI, Axis := v_FeedIndexer); // ML_OpenCyclicPositionChannel
// b_open_channel_FI_done := fb_open_channel_FI.ChannelOpen;

// NETWORK 9
rtrig_reset_open_channel(CLK := b_scc_goto); // R_TRIG
b_open_channel_az R= rtrig_reset_open_channel.Q;
b_open_channel_el R= rtrig_reset_open_channel.Q;
b_open_channel_FI R= rtrig_reset_open_channel.Q;
END_ACTION

ACTION A_StaticPM:
s_mp:= Pointing.StaticPmParameters[Pointing.Status.BandForCorr]; 

// Convert to Radians for trigonometric functions. 
Az_rad:= ML_degtorad(r_write_position_az);
IF r_write_position_el>= 85 THEN
	El_rad:= ML_degtorad(85);
ELSE
	El_rad:= ML_degtorad(r_write_position_el);	
END_IF

ABphi_rad:=ML_degtorad(s_mp.ABphi);

IF Pointing.Status.StaticCorrActive = 1 THEN 
	IF pointing.Status.TiltCorrActive = 1 THEN 
	// Calc Pointing correction with gravity tilt removed
	   TE := 0;
	ELSE 
	// Calc Pointing correction with gravity tilt
	   TE :=1;
    END_IF
	
	 Pointing.Status.StaticPmCorrVal_Az := ( -s_mp.IA - s_mp.CA/COS(El_rad) - s_mp.NPAE*TAN(El_rad) - s_mp.AN*SIN(Az_rad)*TAN(El_rad) - s_mp.AW*COS(Az_rad)*TAN(El_rad) + s_mp.ACEC*COS(Az_rad)
      - s_mp.ACES*SIN(Az_rad) - s_mp.ABA*SIN(ABphi_rad)*COS(2*Az_rad)*(1-TE) +   s_mp.ABA*COS(ABphi_rad)*SIN(2*Az_rad)*(1-TE) + Tracking.Status.act_statOffset_value_Xel/COS(El_rad) +
     (s_mp.AN0*SIN(Az_rad)*TAN(El_rad) + s_mp.AW0*COS(Az_rad)*TAN(El_rad))*TE);
	 
	(* Tiltmeter correction included in static pointing model.
       Pointing.Status.StaticPmCorrVal_Az :=  -s_mp.IA - s_mp.CA/COS(El) - s_mp.NPAE*TAN(El) - s_mp.AN*SIN(Az)*TAN(El) - s_mp.AW*COS(Az)*TAN(El) + s_mp.ACEC*COS(Az)
      - s_mp.ACES*SIN(Az) - s_mp.ABA*SIN(s_mp.ABphi)*COS(2*Az)*(1-TE) +   s_mp.ABA*COS(s_mp.ABphi)*SIN(2*Az)*(1-TE) + Tracking.Status.act_statOffset_value_Xel/COS(El) +
     (ΔAz_tiltmeter + s_mp.AN0*SIN(Az)*TAN(El) + s_mp.AW0*COS(Az)*TAN(El))*TE; *)
	
	Pointing.Status.StaticPmCorrVal_El := (s_mp.IE - s_mp.AN*COS(Az_rad) +s_mp.AW*SIN(Az_rad)+ s_mp.ECEC*COS(El_rad) + s_mp.ECES*SIN(El_rad) + s_mp.ABA*COS(ABphi_rad)*COS(2*Az_rad)*(1-TE) + s_mp.ABA*SIN(ABphi_rad)*SIN(2*Az_rad)*(1-TE) + 
    s_mp.HECE4*COS(4*El_rad) + s_mp.HESE4*SIN(4*El_rad) + s_mp.HECE8*COS(8*El_rad) + s_mp.HESE8*SIN(8*El_rad) + Tracking.Status.act_statOffset_value_El +
    (s_mp.AN0*COS(Az_rad) - s_mp.AW0*SIN(Az_rad))*TE);
	(*  Tiltmeter correction included in static pointing model.
	 Pointing.Status.StaticPmCorrVal_El := s_mp.IE - s_mp.AN*COS(Az) +s_mp.AW*SIN(Az)+ s_mp.ECEC*COS(El) + s_mp.ECES*SIN(El) + s_mp.ABA*COS(s_mp.ABphi)*COS(2*Az)*(1-TE) + s_mp.ABA*SIN(ABphi)*SIN(2*Az)*(1-TE) + 
    s_mp.HECE4*COS(4*El) + s_mp.HESE4*SIN(4*El) + s_mp.HECE8*COS(8*El) + s_mp.HESE8*SIN(8*El) + Tracking.Status.act_statOffset_value_El +
    (ΔEl_tiltmeter + s_mp.AN0*COS(Az) - s_mp.AW0*SIN(Az))*TE; *)
   
ELSE 
// No calculation of static model only offsets
   Pointing.Status.StaticPmCorrVal_Az := (Tracking.Status.act_statOffset_value_Xel/COS(El_rad));
   Pointing.Status.StaticPmCorrVal_El := Tracking.Status.act_statOffset_value_El;
END_IF


IF   ABS(Pointing.Status.StaticPmCorrVal_Az) > gc_lr_point_corr_error_lim OR  ABS(Pointing.Status.StaticPmCorrVal_El) > gc_lr_point_corr_error_lim THEN 
   Pointing.Status.StaticPmCorrVal_Az := 0; 
   Pointing.Status.StaticPmCorrVal_El := 0;
   Management.ErrorStatus.errPoint := 1; 
END_IF
END_ACTION

ACTION A_DynamicPM:
	IF Pointing.Status.TiltOne_On THEN 
    	Pointing.Status.TiltCorrVal_Az:= Pointing.Status.TiltYArcsec_One*TAN(El_rad); //El_rad is calculated in the Stati PM section 
		Pointing.Status.TiltCorrVal_El:= Pointing.Status.TiltXArcsec_One;
	ELSIF Pointing.Status.TiltTwo_On THEN
		Pointing.Status.TiltCorrVal_Az:= Pointing.Status.TiltYArcsec_One*TAN(El_rad);
		Pointing.Status.TiltCorrVal_El:= Pointing.Status.TiltXArcsec_One;
	ELSE
		Pointing.Status.TiltCorrVal_Az:= 0;
		Pointing.Status.TiltCorrVal_El:= 0;
	END_IF

//	Check velocity
IF  ABS(axisdata[1].rActualVelocity_i)>= gc_r_tilt_vel_limit_Az THEN 
	Pointing.Status.TiltCorrVal_Az:= 0;
    Pointing.Status.TiltCorrVal_El:= 0;
END_IF

// Check if the correction is with in limits 
// The behaviour if the correction is outside the limits still needs to be finalised
IF ABS(Pointing.Status.TiltCorrVal_Az)>= gc_lr_tilt_corr_limit_Az OR ABS(Pointing.Status.TiltCorrVal_El)>=gc_lr_tilt_corr_limit_El THEN 
	Pointing.Status.TiltCorrVal_Az:= gc_lr_tilt_corr_limit_Az;
    Pointing.Status.TiltCorrVal_El:= gc_lr_tilt_corr_limit_El;
END_IF
END_ACTION

ACTION A_AmbTempPM:
IF Pointing.Status.AmbTempCorrActive THEN 
	Pointing.Status.AmbTempCorrVal_Az:=0;
	Pointing.Status.AmbTempCorrVal_El:=0;
ELSE
	Pointing.Status.AmbTempCorrVal_Az:=0;
	Pointing.Status.AmbTempCorrVal_El:=0;
END_IF
END_ACTION

ACTION A_Sim_track_function_blocks:
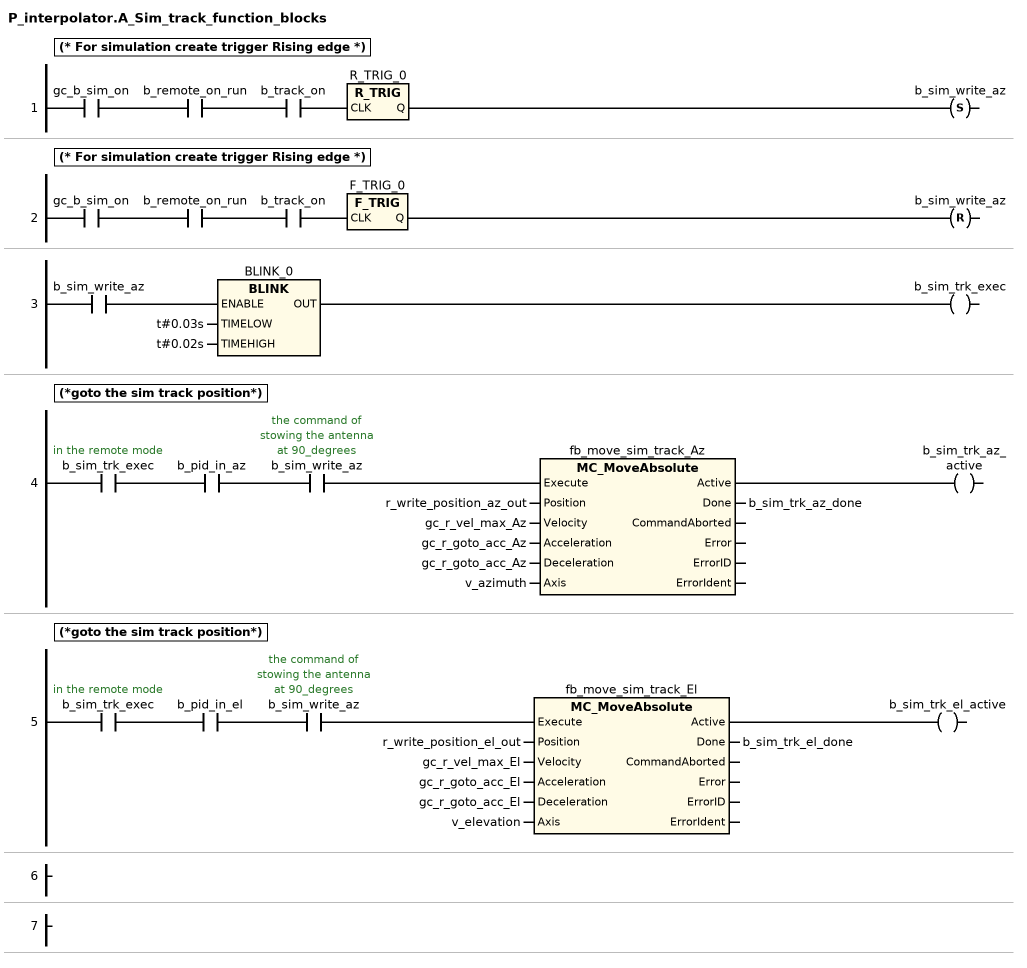
// NETWORK 1
// label: (* For simulation create trigger Rising edge *)
R_TRIG_0(CLK := gc_b_sim_on AND b_remote_on_run AND b_track_on); // R_TRIG
b_sim_write_az S= R_TRIG_0.Q;

// NETWORK 2
// label: (* For simulation create trigger Rising edge *)
F_TRIG_0(CLK := gc_b_sim_on AND b_remote_on_run AND b_track_on); // F_TRIG
b_sim_write_az R= F_TRIG_0.Q;

// NETWORK 3
BLINK_0(ENABLE := b_sim_write_az, TIMELOW := t#0.03s, TIMEHIGH := t#0.02s); // BLINK
b_sim_trk_exec := BLINK_0.OUT;

// NETWORK 4
//   fb_move_sim_track_Az: move the elevation to the fixed position
//   b_sim_trk_exec: in the remote mode
//   b_sim_write_az: the command of stowing the antenna at 90_degrees
//   v_azimuth: Virtual axis "v_elevation" with axis number 8
// label: (*goto the sim track position*)
fb_move_sim_track_Az(
    Execute := b_sim_trk_exec AND b_pid_in_az AND b_sim_write_az,
    Position := r_write_position_az_out,
    Velocity := gc_r_vel_max_Az,
    Acceleration := gc_r_goto_acc_Az,
    Deceleration := gc_r_goto_acc_Az,
    Axis := v_azimuth,
    Done => b_sim_trk_az_done); // MC_MoveAbsolute
b_sim_trk_az_active := fb_move_sim_track_Az.Active;

// NETWORK 5
//   fb_move_sim_track_El: move the elevation to the fixed position
//   b_sim_trk_exec: in the remote mode
//   b_sim_write_az: the command of stowing the antenna at 90_degrees
//   v_elevation: Virtual axis "v_elevation" with axis number 8
// label: (*goto the sim track position*)
fb_move_sim_track_El(
    Execute := b_sim_trk_exec AND b_pid_in_el AND b_sim_write_az,
    Position := r_write_position_el_out,
    Velocity := gc_r_vel_max_El,
    Acceleration := gc_r_goto_acc_El,
    Deceleration := gc_r_goto_acc_El,
    Axis := v_elevation,
    Done => b_sim_trk_el_done); // MC_MoveAbsolute
b_sim_trk_el_active := fb_move_sim_track_El.Active;

// NETWORK 6

// NETWORK 7
END_ACTION

END_PROGRAM

// IndraMotionMlc1/Application/POUs/Panel Function/FI_TEST
PROGRAM FI_TEST
VAR
	MC_Power_0: MC_Power;
	fi_enable1: BOOL;
	MC_Power_1: MC_Power;
	fi_enable2: BOOL;
	MC_TorqueControl_0: MC_TorqueControl;
	fi_torque1: BOOL;
	MC_TorqueControl_1: MC_TorqueControl;
	fi_torque2: BOOL;
	MC_MoveVelocity_0: MC_MoveVelocity;
	fi_move1: BOOL;
	fi_vel1: REAL;
	BLINK_0: BLINK;
	BLINK_1: BLINK;
	MC_MoveVelocity_1: MC_MoveVelocity;
	fi_move2: BOOL;
	fi_vel2: REAL;
	BLINK_2: BLINK;
	MB_ReadRealParameter_0: MB_ReadRealParameter;
	fi_encoder1: REAL;
	MB_ReadRealParameter_1: MB_ReadRealParameter;
	fi_encoder2: REAL;
	MC_Stop_0: MC_Stop;
	MC_Stop_1: MC_Stop;
	fi_stop: BOOL;
	R_TRIG_0: R_TRIG;
	R_TRIG_1: R_TRIG;
	R_TRIG_2: R_TRIG;
	R_TRIG_3: R_TRIG;
	MB_ReadParameter_0: MB_ReadParameter;
	MB_ReadParameter_1: MB_ReadParameter;
	fi_brake1: DWORD;
	fi_brake2: DWORD;
END_VAR

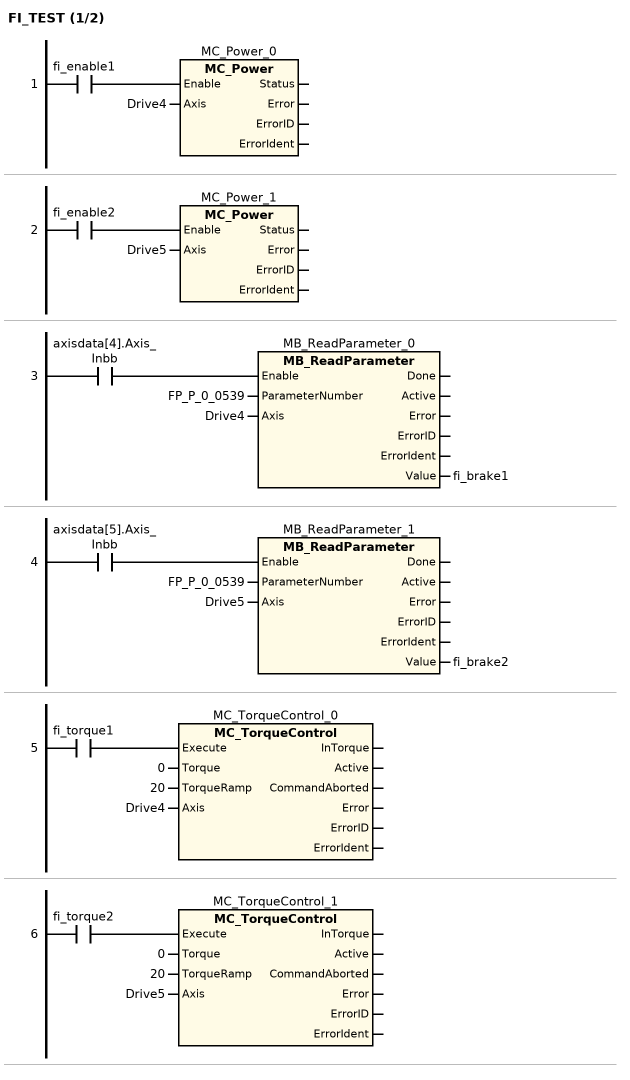
// NETWORK 1
MC_Power_0(Enable := fi_enable1, Axis := Drive4); // MC_Power

// NETWORK 2
MC_Power_1(Enable := fi_enable2, Axis := Drive5); // MC_Power

// NETWORK 3
MB_ReadParameter_0(
    Enable := axisdata[4].Axis_Inbb,
    ParameterNumber := FP_P_0_0539,
    Axis := Drive4,
    Value => fi_brake1); // MB_ReadParameter

// NETWORK 4
MB_ReadParameter_1(
    Enable := axisdata[5].Axis_Inbb,
    ParameterNumber := FP_P_0_0539,
    Axis := Drive5,
    Value => fi_brake2); // MB_ReadParameter

// NETWORK 5
MC_TorqueControl_0(Execute := fi_torque1, Torque := 0, TorqueRamp := 20, Axis := Drive4); // MC_TorqueControl

// NETWORK 6
MC_TorqueControl_1(Execute := fi_torque2, Torque := 0, TorqueRamp := 20, Axis := Drive5); // MC_TorqueControl

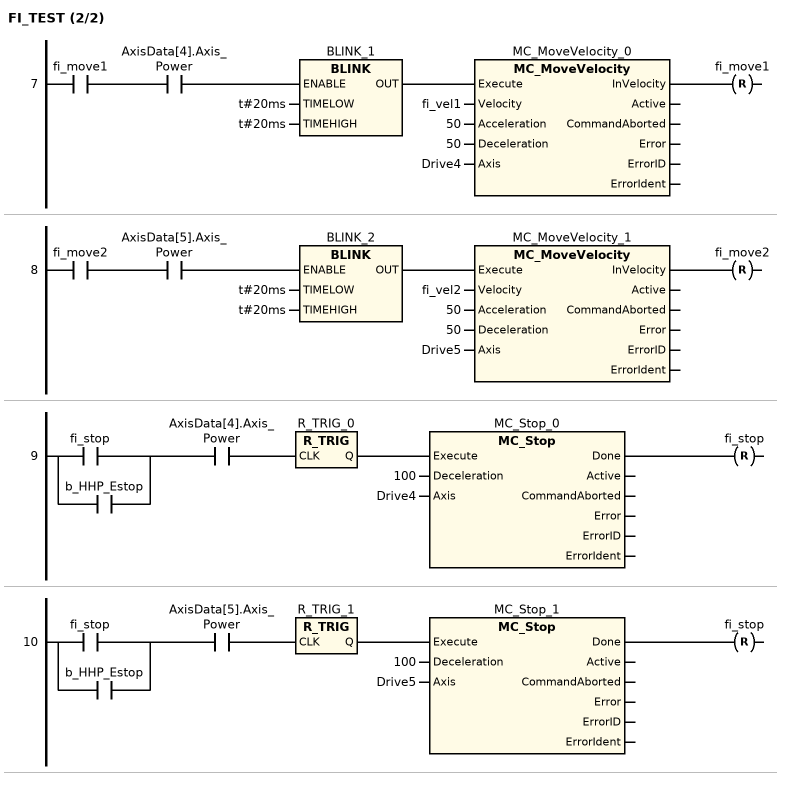
// NETWORK 7
BLINK_1(ENABLE := fi_move1 AND AxisData[4].Axis_Power, TIMELOW := t#20ms, TIMEHIGH := t#20ms); // BLINK
MC_MoveVelocity_0(
    Execute := BLINK_1.OUT,
    Velocity := fi_vel1,
    Acceleration := 50,
    Deceleration := 50,
    Axis := Drive4); // MC_MoveVelocity
fi_move1 R= MC_MoveVelocity_0.InVelocity;

// NETWORK 8
BLINK_2(ENABLE := fi_move2 AND AxisData[5].Axis_Power, TIMELOW := t#20ms, TIMEHIGH := t#20ms); // BLINK
MC_MoveVelocity_1(
    Execute := BLINK_2.OUT,
    Velocity := fi_vel2,
    Acceleration := 50,
    Deceleration := 50,
    Axis := Drive5); // MC_MoveVelocity
fi_move2 R= MC_MoveVelocity_1.InVelocity;

// NETWORK 9
R_TRIG_0(CLK := (fi_stop OR b_HHP_Estop) AND AxisData[4].Axis_Power); // R_TRIG
MC_Stop_0(Execute := R_TRIG_0.Q, Deceleration := 100, Axis := Drive4); // MC_Stop
fi_stop R= MC_Stop_0.Done;

// NETWORK 10
R_TRIG_1(CLK := (fi_stop OR b_HHP_Estop) AND AxisData[5].Axis_Power); // R_TRIG
MC_Stop_1(Execute := R_TRIG_1.Q, Deceleration := 100, Axis := Drive5); // MC_Stop
fi_stop R= MC_Stop_1.Done;

END_PROGRAM

// IndraMotionMlc1/Application/POUs/Panel Function/LOCK_TEST
PROGRAM LOCK_TEST
VAR
	lock_enable: BOOL;
	unlock_enable: BOOL;
	power_on: BOOL;
	el_enable: BOOL;
	b_move: BOOL;
	stop_enable: BOOL;
	MC_MoveVelocity_0: MC_MoveVelocity;
	MC_Power_0: MC_Power;
	vel_el: REAL;
	
	MC_Stop_0: MC_Stop;
	R_TRIG_0: R_TRIG;
	R_TRIG_1: R_TRIG;
	MB_ReadRealParameter_0: MB_ReadRealParameter;
	el_motorencoder: REAL;
	up_limit: BOOL;
	down_limit: BOOL;
	down_stop: BOOL;
	up_stop: BOOL;
	MC_MoveVelocity_1: MC_MoveVelocity;
	R_TRIG_2: R_TRIG;
	clear_error: BOOL;
	
	ML_WriteParameter_0: ML_WriteParameter;
	R_TRIG_3: R_TRIG;
	TON_0: TON;
	vel_run:BOOL;
	el_enable1:BOOL;
	
	R_TRIG_4: R_TRIG;
	R_TRIG_5: R_TRIG;
	FB_clear_error_1: MB_WriteParameter;
	TON_1: TON;
	R_TRIG_6: R_TRIG;
	R_TRIG_7: R_TRIG;
	R_TRIG_8: R_TRIG;
	BLINK_0: BLINK;
	R_TRIG_9: R_TRIG;
	R_TRIG_10: R_TRIG;
	MC_MoveVelocity_2: MC_MoveVelocity;
	R_TRIG_11: R_TRIG;
	MC_Power_1: MC_Power;
	az_enable: BOOL;
	BLINK_1: BLINK;
	MC_MoveVelocity_3: MC_MoveVelocity;
	b_move2: BOOL;
	vel_az: LREAL;
	MB_ReadRealParameter_1: MB_ReadRealParameter;
	az_motorencoder: REAL;
	MC_Power_2: MC_Power;
	az_enable2: BOOL;
	MC_TorqueControl_0: MC_TorqueControl;
	b_torque_1: BOOL;
	MC_TorqueControl_1: MC_TorqueControl;
	b_torque_2: BOOL;
	BLINK_2: BLINK;
	MC_MoveVelocity_4: MC_MoveVelocity;
	b_move3: BOOL;
	ccw_limit: BOOL;
	ccw_stop: BOOL;
	cw_limit: BOOL;
	cw_stop: BOOL;
	MC_MoveVelocity_5: MC_MoveVelocity;
	R_TRIG_12: R_TRIG;
	MC_MoveVelocity_6: MC_MoveVelocity;
	R_TRIG_13: R_TRIG;
	MC_MoveVelocity_7: MC_MoveVelocity;
	R_TRIG_14: R_TRIG;
	MC_MoveVelocity_8: MC_MoveVelocity;
	BLINK_3: BLINK;
	R_TRIG_15: R_TRIG;
	MC_Stop_1: MC_Stop;
	MC_Stop_2: MC_Stop;
	stop_enable1: BOOL;
	R_TRIG_16: R_TRIG;
	R_TRIG_17: R_TRIG;
	MC_MoveAbsolute_0: MC_MoveAbsolute;
	el_pos: BOOL;
	R_TRIG_18: R_TRIG;
	el_pos_cmd: REAL;
	MC_MoveAbsolute_1: MC_MoveAbsolute;
	R_TRIG_19: R_TRIG;
	MC_MoveAbsolute_2: MC_MoveAbsolute;
	R_TRIG_20: R_TRIG;
	az_pos: BOOL;
	az_angle: REAL;
	az_vel: REAL;
	stop_enable2: BOOL;
	R_TRIG_21: R_TRIG;
	az_enable1: BOOL;	
	az2_enable: BOOL;
	az1_enable: BOOL;
	MC_Power_3: MC_Power;
	TON_2: TON;
	MC_Power_4: MC_Power;
	TON_3: TON;
	az_enable_step1: BOOL;
	MC_MoveAbsolute_3: MC_MoveAbsolute;
	az_enable_step2: BOOL;
	MB_GearInPos_0: MB_GearInPos;
	TON_4: TON;
	MC_Stop_3: MC_Stop;
	R_TRIG_22: R_TRIG;
	R_TRIG_23: R_TRIG;
	az_disable: BOOL;
	MC_GearOut_0: MC_GearOut;
	MC_Stop_4: MC_Stop;
	R_TRIG_24: R_TRIG;
	R_TRIG_25: R_TRIG;
	R_TRIG_26: R_TRIG;
	MC_GearOut_1: MC_GearOut;
	MC_Stop_5: MC_Stop;
	R_TRIG_27: R_TRIG;
	R_TRIG_28: R_TRIG;
	R_TRIG_29: R_TRIG;
	TON_5: TON;
	R_TRIG_30: R_TRIG;
	MC_MoveAbsolute_4: MC_MoveAbsolute;
	BLINK_4: BLINK;
	MC_MoveVelocity_9: MC_MoveVelocity;
	R_TRIG_31: R_TRIG;
	MC_MoveVelocity_10: MC_MoveVelocity;
	R_TRIG_32: R_TRIG;
	MC_MoveVelocity_11: MC_MoveVelocity;
	R_TRIG_33: R_TRIG;
	MC_Stop_6: MC_Stop;
	stop_enable_az: BOOL;
	enable_bottom: BOOL;
	disable_bottom: BOOL;
	stow_bottom: BOOL;
	cw_bottom: BOOL;
	ccw_bottom: BOOL;
	reset_bottom: BOOL;
	R_TRIG_34: R_TRIG;
	dance_enable: BOOL;
	R_TRIG_35: R_TRIG;
	dance_enable_az1: BOOL;
	dance_enable_az2: BOOL;
	dance_enable_el: BOOL;
	dance_disable_az: BOOL;
	MC_TorqueControl_2: MC_TorqueControl;
	el_torque1: BOOL;
	torque_test: REAL;
	az_pos_test: REAL;
END_VAR
VAR // added by the converter: edge detectors and wires of the graphical bodies
    _w1 : BOOL;
END_VAR

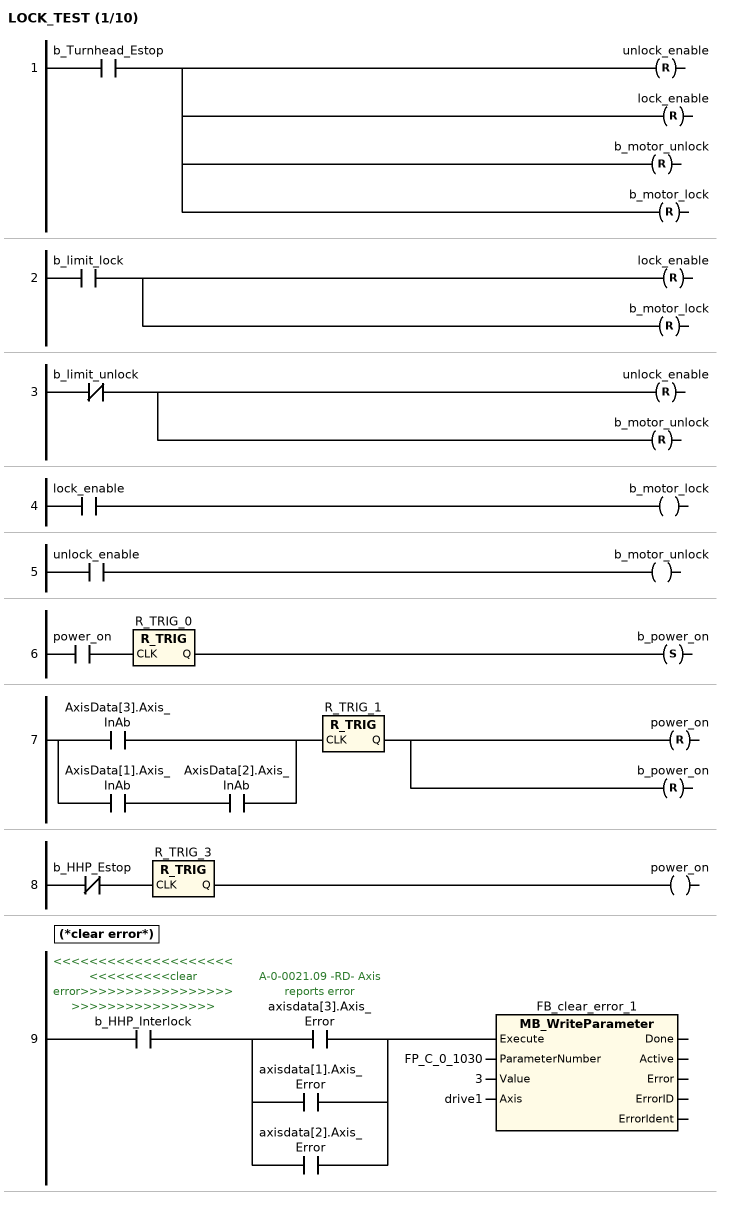
// NETWORK 1
unlock_enable R= b_Turnhead_Estop;
lock_enable R= b_Turnhead_Estop;
b_motor_unlock R= b_Turnhead_Estop;
b_motor_lock R= b_Turnhead_Estop;

// NETWORK 2
lock_enable R= b_limit_lock;
b_motor_lock R= b_limit_lock;

// NETWORK 3
_w1 := NOT b_limit_unlock;
unlock_enable R= _w1;
b_motor_unlock R= _w1;

// NETWORK 4
b_motor_lock := lock_enable;

// NETWORK 5
b_motor_unlock := unlock_enable;

// NETWORK 6
R_TRIG_0(CLK := power_on); // R_TRIG
b_power_on S= R_TRIG_0.Q;

// NETWORK 7
R_TRIG_1(CLK := AxisData[3].Axis_InAb OR AxisData[1].Axis_InAb AND AxisData[2].Axis_InAb); // R_TRIG
power_on R= R_TRIG_1.Q;
b_power_on R= R_TRIG_1.Q;

// NETWORK 8
R_TRIG_3(CLK := NOT b_HHP_Estop); // R_TRIG
power_on := R_TRIG_3.Q;

// NETWORK 9
//   b_HHP_Interlock: <<<<<<<<<<<<<<<<<<<<<<<<<<<<<clear error>>>>>>>>>>>>>>>>>>>>>>>>>>>>>>>>>
//   axisdata[3].Axis_Error: A-0-0021.09 -RD- Axis reports error
//   FP_C_0_1030: Command: Clear all control errors
//   drive1: Real axis "Drive1" with axis number 1
// label: (*clear error*)
FB_clear_error_1(
    Execute := b_HHP_Interlock AND (axisdata[3].Axis_Error OR axisdata[1].Axis_Error OR axisdata[2].Axis_Error),
    ParameterNumber := FP_C_0_1030,
    Value := 3,
    Axis := drive1); // MB_WriteParameter

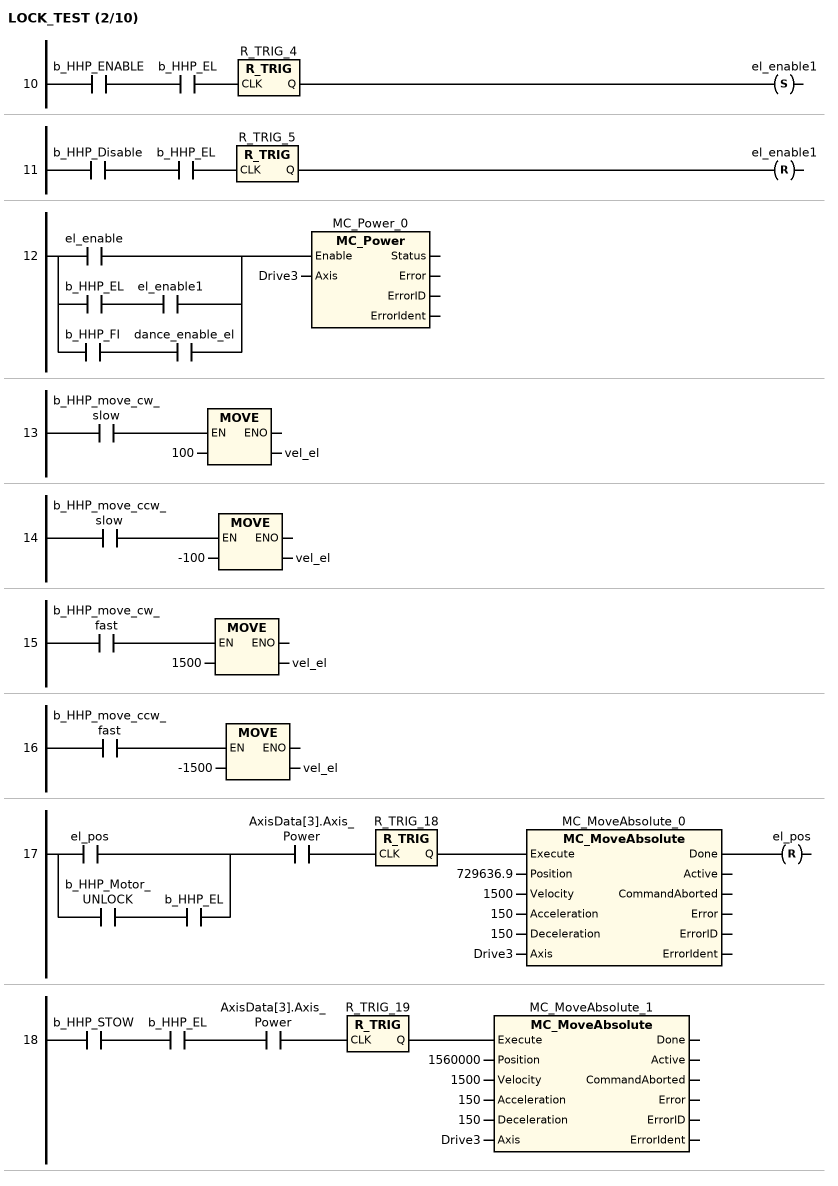
// NETWORK 10
R_TRIG_4(CLK := b_HHP_ENABLE AND b_HHP_EL); // R_TRIG
el_enable1 S= R_TRIG_4.Q;

// NETWORK 11
R_TRIG_5(CLK := b_HHP_Disable AND b_HHP_EL); // R_TRIG
el_enable1 R= R_TRIG_5.Q;

// NETWORK 12
MC_Power_0(Enable := el_enable OR b_HHP_EL AND el_enable1 OR b_HHP_FI AND dance_enable_el, Axis := Drive3); // MC_Power

// NETWORK 13
IF b_HHP_move_cw_slow THEN vel_el := 100; END_IF

// NETWORK 14
IF b_HHP_move_ccw_slow THEN vel_el := -100; END_IF

// NETWORK 15
IF b_HHP_move_cw_fast THEN vel_el := 1500; END_IF

// NETWORK 16
IF b_HHP_move_ccw_fast THEN vel_el := -1500; END_IF

// NETWORK 17
R_TRIG_18(CLK := (el_pos OR b_HHP_Motor_UNLOCK AND b_HHP_EL) AND AxisData[3].Axis_Power); // R_TRIG
MC_MoveAbsolute_0(
    Execute := R_TRIG_18.Q,
    Position := 729636.9,
    Velocity := 1500,
    Acceleration := 150,
    Deceleration := 150,
    Axis := Drive3); // MC_MoveAbsolute
el_pos R= MC_MoveAbsolute_0.Done;

// NETWORK 18
R_TRIG_19(CLK := b_HHP_STOW AND b_HHP_EL AND AxisData[3].Axis_Power); // R_TRIG
MC_MoveAbsolute_1(
    Execute := R_TRIG_19.Q,
    Position := 1560000,
    Velocity := 1500,
    Acceleration := 150,
    Deceleration := 150,
    Axis := Drive3); // MC_MoveAbsolute

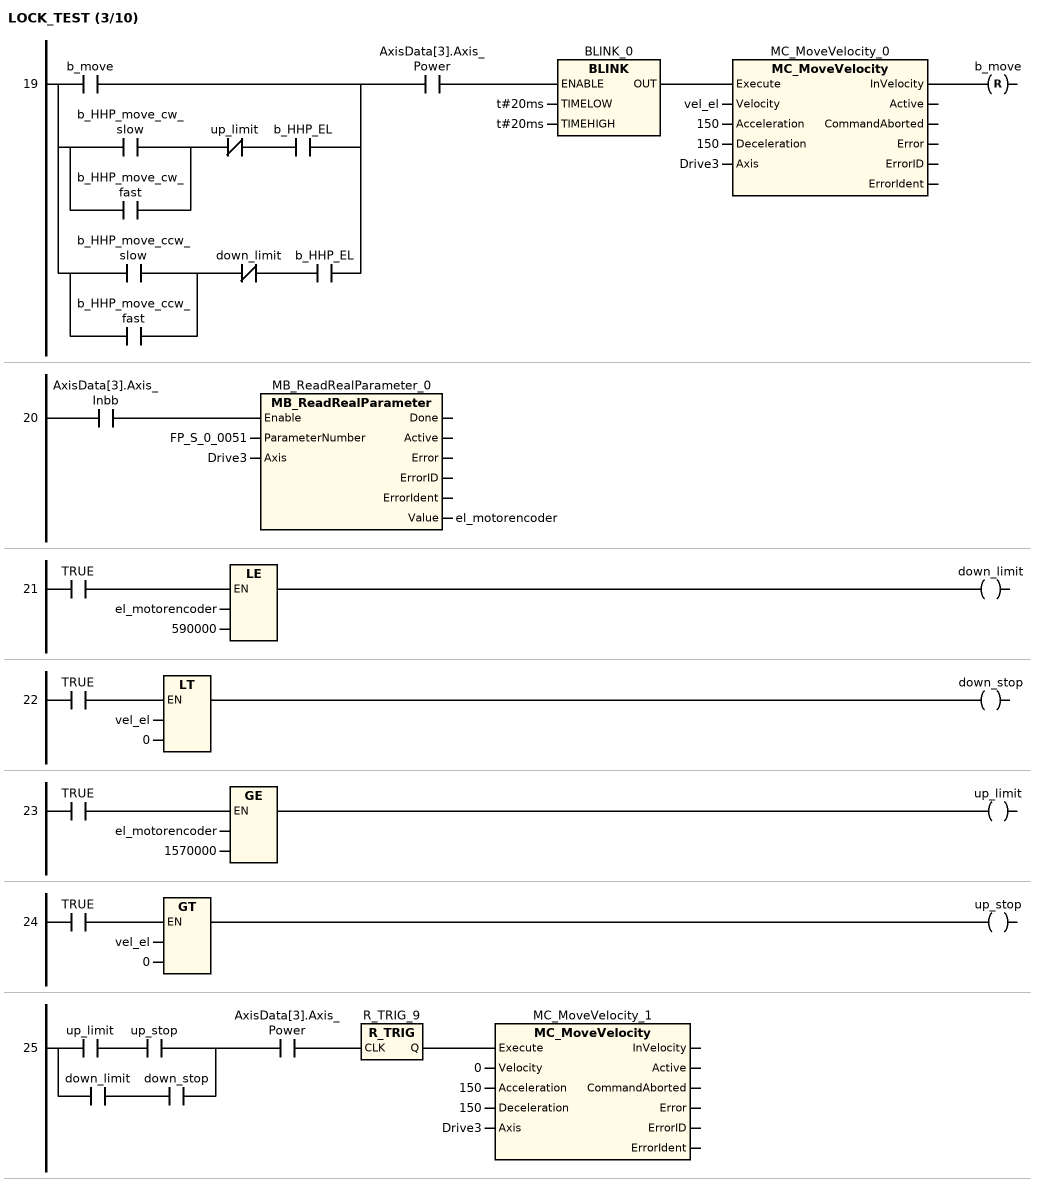
// NETWORK 19
BLINK_0(
    ENABLE := (b_move OR (b_HHP_move_cw_slow OR b_HHP_move_cw_fast) AND NOT up_limit AND b_HHP_EL OR (b_HHP_move_ccw_slow OR b_HHP_move_ccw_fast) AND NOT down_limit AND b_HHP_EL) AND AxisData[3].Axis_Power,
    TIMELOW := t#20ms,
    TIMEHIGH := t#20ms); // BLINK
MC_MoveVelocity_0(
    Execute := BLINK_0.OUT,
    Velocity := vel_el,
    Acceleration := 150,
    Deceleration := 150,
    Axis := Drive3); // MC_MoveVelocity
b_move R= MC_MoveVelocity_0.InVelocity;

// NETWORK 20
MB_ReadRealParameter_0(
    Enable := AxisData[3].Axis_Inbb,
    ParameterNumber := FP_S_0_0051,
    Axis := Drive3,
    Value => el_motorencoder); // MB_ReadRealParameter

// NETWORK 21
down_limit := el_motorencoder <= 590000;

// NETWORK 22
down_stop := vel_el < 0;

// NETWORK 23
up_limit := el_motorencoder >= 1570000;

// NETWORK 24
up_stop := vel_el > 0;

// NETWORK 25
R_TRIG_9(CLK := (up_limit AND up_stop OR down_limit AND down_stop) AND AxisData[3].Axis_Power); // R_TRIG
MC_MoveVelocity_1(
    Execute := R_TRIG_9.Q,
    Velocity := 0,
    Acceleration := 150,
    Deceleration := 150,
    Axis := Drive3); // MC_MoveVelocity

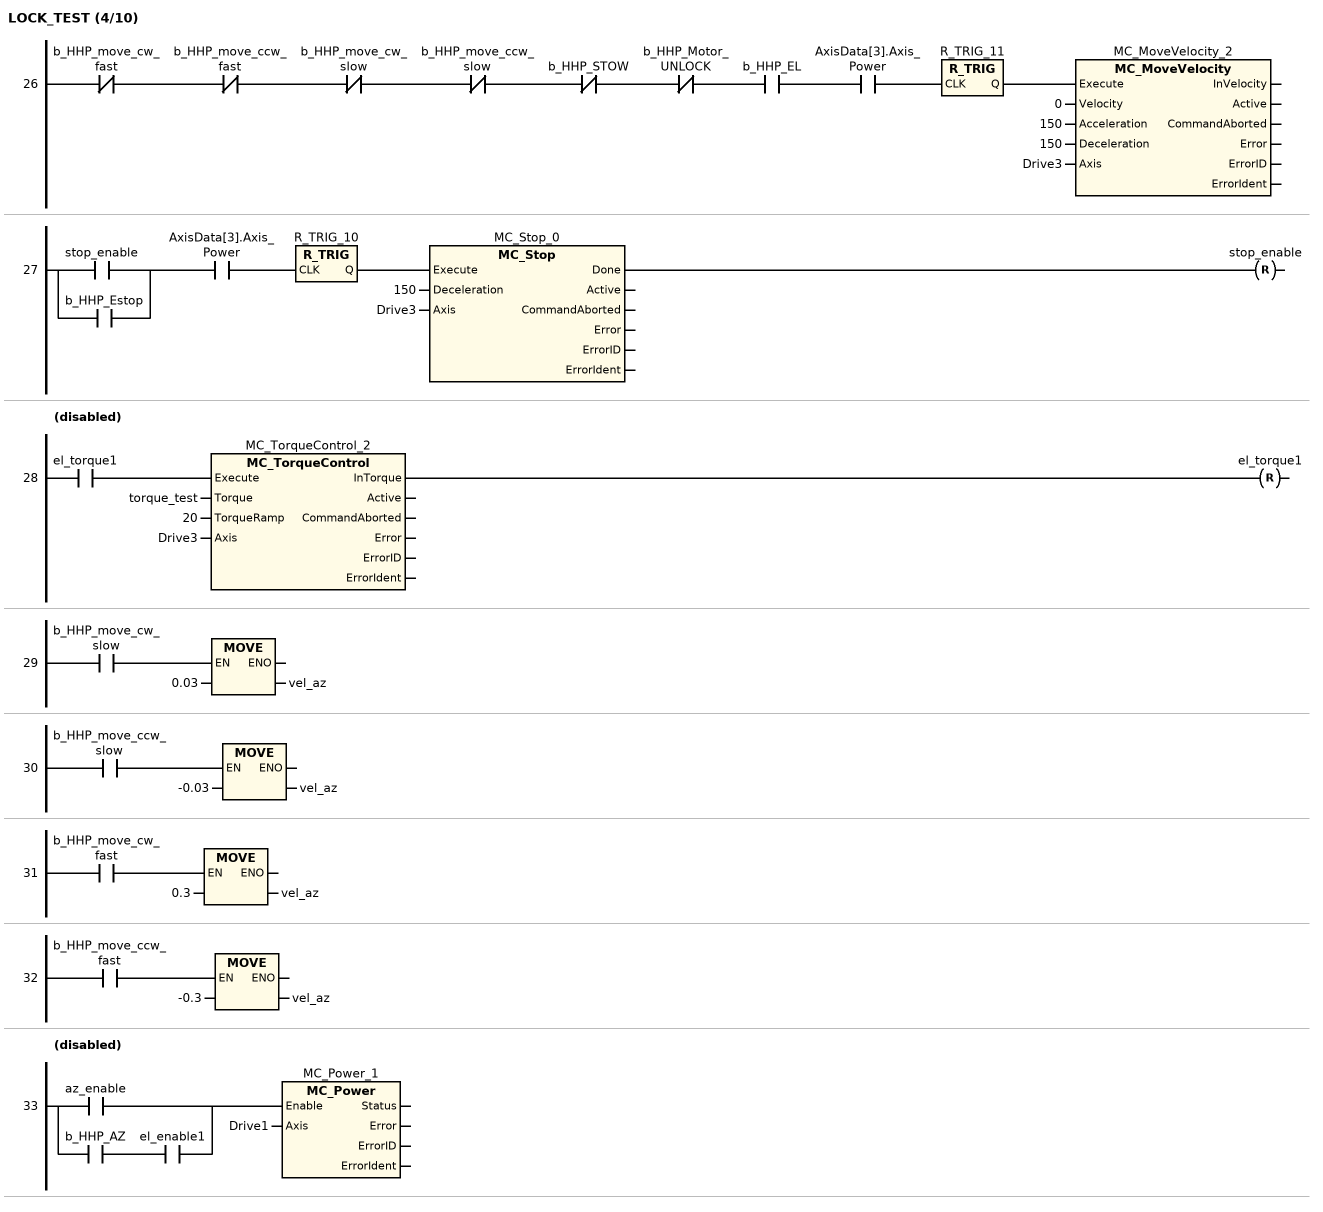
// NETWORK 26
R_TRIG_11(CLK := NOT b_HHP_move_cw_fast AND NOT b_HHP_move_ccw_fast AND NOT b_HHP_move_cw_slow AND NOT b_HHP_move_ccw_slow AND NOT b_HHP_STOW AND NOT b_HHP_Motor_UNLOCK AND b_HHP_EL AND AxisData[3].Axis_Power); // R_TRIG
MC_MoveVelocity_2(
    Execute := R_TRIG_11.Q,
    Velocity := 0,
    Acceleration := 150,
    Deceleration := 150,
    Axis := Drive3); // MC_MoveVelocity

// NETWORK 27
R_TRIG_10(CLK := (stop_enable OR b_HHP_Estop) AND AxisData[3].Axis_Power); // R_TRIG
MC_Stop_0(Execute := R_TRIG_10.Q, Deceleration := 150, Axis := Drive3); // MC_Stop
stop_enable R= MC_Stop_0.Done;

// NETWORK 28 (disabled)
// MC_TorqueControl_2(Execute := el_torque1, Torque := torque_test, TorqueRamp := 20, Axis := Drive3); // MC_TorqueControl
// el_torque1 R= MC_TorqueControl_2.InTorque;

// NETWORK 29
IF b_HHP_move_cw_slow THEN vel_az := 0.03; END_IF

// NETWORK 30
IF b_HHP_move_ccw_slow THEN vel_az := -0.03; END_IF

// NETWORK 31
IF b_HHP_move_cw_fast THEN vel_az := 0.3; END_IF

// NETWORK 32
IF b_HHP_move_ccw_fast THEN vel_az := -0.3; END_IF

// NETWORK 33 (disabled)
// MC_Power_1(Enable := az_enable OR b_HHP_AZ AND el_enable1, Axis := Drive1); // MC_Power

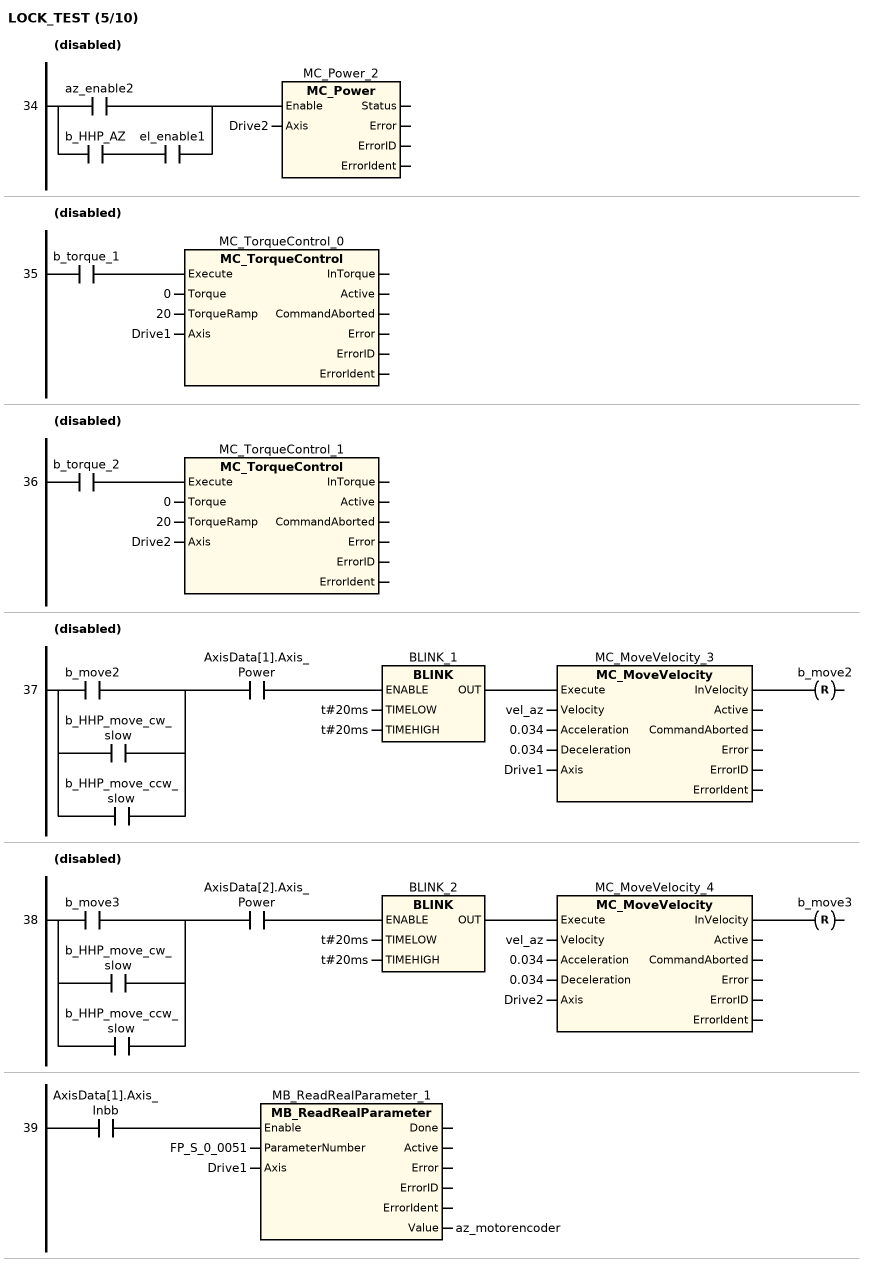
// NETWORK 34 (disabled)
// MC_Power_2(Enable := az_enable2 OR b_HHP_AZ AND el_enable1, Axis := Drive2); // MC_Power

// NETWORK 35 (disabled)
// MC_TorqueControl_0(Execute := b_torque_1, Torque := 0, TorqueRamp := 20, Axis := Drive1); // MC_TorqueControl

// NETWORK 36 (disabled)
// MC_TorqueControl_1(Execute := b_torque_2, Torque := 0, TorqueRamp := 20, Axis := Drive2); // MC_TorqueControl

// NETWORK 37 (disabled)
// BLINK_1(
//     ENABLE := (b_move2 OR b_HHP_move_cw_slow OR b_HHP_move_ccw_slow) AND AxisData[1].Axis_Power,
//     TIMELOW := t#20ms,
//     TIMEHIGH := t#20ms); // BLINK
// MC_MoveVelocity_3(
//     Execute := BLINK_1.OUT,
//     Velocity := vel_az,
//     Acceleration := 0.034,
//     Deceleration := 0.034,
//     Axis := Drive1); // MC_MoveVelocity
// b_move2 R= MC_MoveVelocity_3.InVelocity;

// NETWORK 38 (disabled)
// BLINK_2(
//     ENABLE := (b_move3 OR b_HHP_move_cw_slow OR b_HHP_move_ccw_slow) AND AxisData[2].Axis_Power,
//     TIMELOW := t#20ms,
//     TIMEHIGH := t#20ms); // BLINK
// MC_MoveVelocity_4(
//     Execute := BLINK_2.OUT,
//     Velocity := vel_az,
//     Acceleration := 0.034,
//     Deceleration := 0.034,
//     Axis := Drive2); // MC_MoveVelocity
// b_move3 R= MC_MoveVelocity_4.InVelocity;

// NETWORK 39
MB_ReadRealParameter_1(
    Enable := AxisData[1].Axis_Inbb,
    ParameterNumber := FP_S_0_0051,
    Axis := Drive1,
    Value => az_motorencoder); // MB_ReadRealParameter

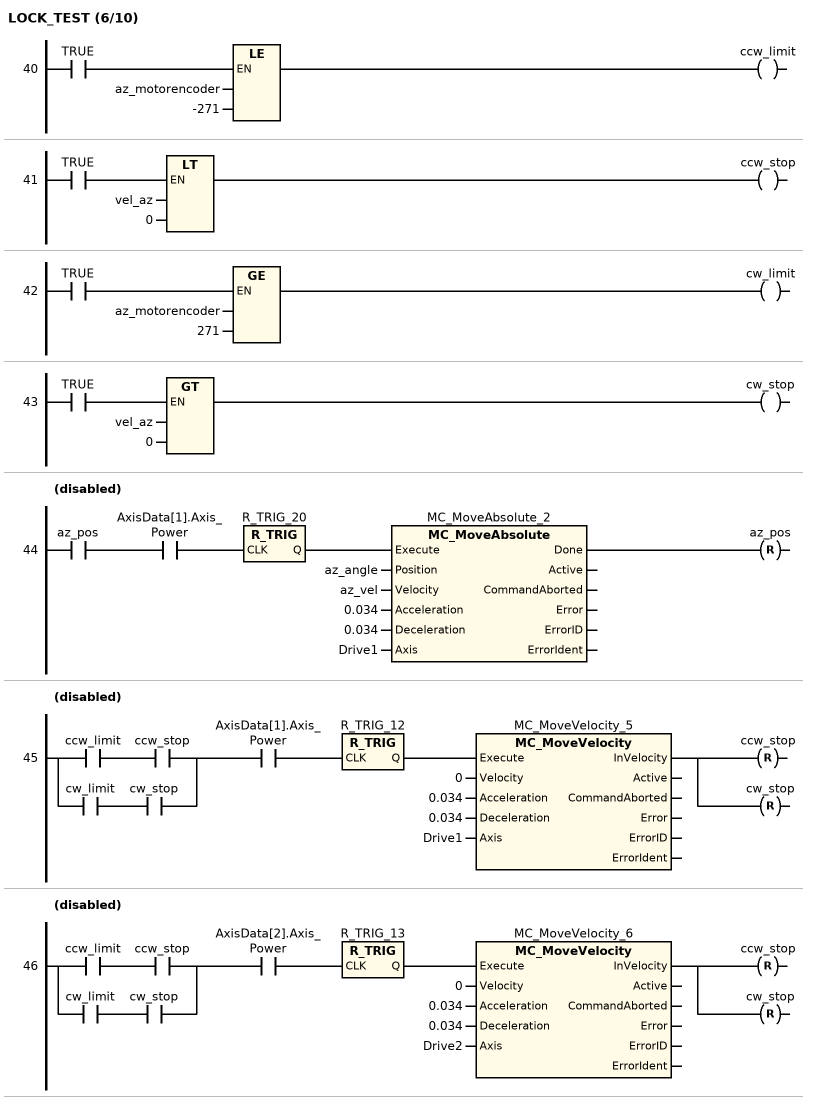
// NETWORK 40
ccw_limit := az_motorencoder <= -271;

// NETWORK 41
ccw_stop := vel_az < 0;

// NETWORK 42
cw_limit := az_motorencoder >= 271;

// NETWORK 43
cw_stop := vel_az > 0;

// NETWORK 44 (disabled)
// R_TRIG_20(CLK := az_pos AND AxisData[1].Axis_Power); // R_TRIG
// MC_MoveAbsolute_2(
//     Execute := R_TRIG_20.Q,
//     Position := az_angle,
//     Velocity := az_vel,
//     Acceleration := 0.034,
//     Deceleration := 0.034,
//     Axis := Drive1); // MC_MoveAbsolute
// az_pos R= MC_MoveAbsolute_2.Done;

// NETWORK 45 (disabled)
// R_TRIG_12(CLK := (ccw_limit AND ccw_stop OR cw_limit AND cw_stop) AND AxisData[1].Axis_Power); // R_TRIG
// MC_MoveVelocity_5(
//     Execute := R_TRIG_12.Q,
//     Velocity := 0,
//     Acceleration := 0.034,
//     Deceleration := 0.034,
//     Axis := Drive1); // MC_MoveVelocity
// ccw_stop R= MC_MoveVelocity_5.InVelocity;
// cw_stop R= MC_MoveVelocity_5.InVelocity;

// NETWORK 46 (disabled)
// R_TRIG_13(CLK := (ccw_limit AND ccw_stop OR cw_limit AND cw_stop) AND AxisData[2].Axis_Power); // R_TRIG
// MC_MoveVelocity_6(
//     Execute := R_TRIG_13.Q,
//     Velocity := 0,
//     Acceleration := 0.034,
//     Deceleration := 0.034,
//     Axis := Drive2); // MC_MoveVelocity
// ccw_stop R= MC_MoveVelocity_6.InVelocity;
// cw_stop R= MC_MoveVelocity_6.InVelocity;

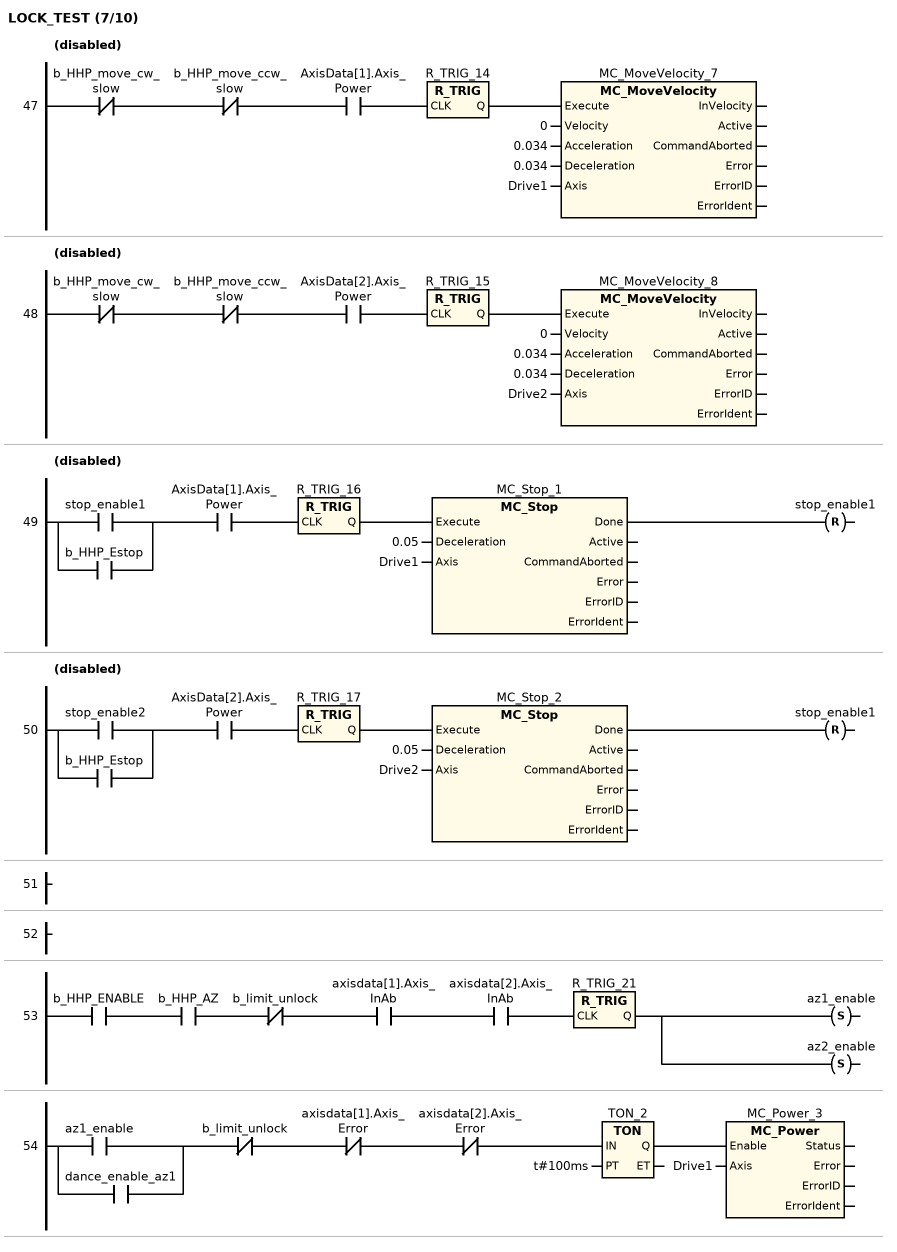
// NETWORK 47 (disabled)
// R_TRIG_14(CLK := NOT b_HHP_move_cw_slow AND NOT b_HHP_move_ccw_slow AND AxisData[1].Axis_Power); // R_TRIG
// MC_MoveVelocity_7(
//     Execute := R_TRIG_14.Q,
//     Velocity := 0,
//     Acceleration := 0.034,
//     Deceleration := 0.034,
//     Axis := Drive1); // MC_MoveVelocity

// NETWORK 48 (disabled)
// R_TRIG_15(CLK := NOT b_HHP_move_cw_slow AND NOT b_HHP_move_ccw_slow AND AxisData[2].Axis_Power); // R_TRIG
// MC_MoveVelocity_8(
//     Execute := R_TRIG_15.Q,
//     Velocity := 0,
//     Acceleration := 0.034,
//     Deceleration := 0.034,
//     Axis := Drive2); // MC_MoveVelocity

// NETWORK 49 (disabled)
// R_TRIG_16(CLK := (stop_enable1 OR b_HHP_Estop) AND AxisData[1].Axis_Power); // R_TRIG
// MC_Stop_1(Execute := R_TRIG_16.Q, Deceleration := 0.05, Axis := Drive1); // MC_Stop
// stop_enable1 R= MC_Stop_1.Done;

// NETWORK 50 (disabled)
// R_TRIG_17(CLK := (stop_enable2 OR b_HHP_Estop) AND AxisData[2].Axis_Power); // R_TRIG
// MC_Stop_2(Execute := R_TRIG_17.Q, Deceleration := 0.05, Axis := Drive2); // MC_Stop
// stop_enable1 R= MC_Stop_2.Done;

// NETWORK 51

// NETWORK 52

// NETWORK 53
R_TRIG_21(CLK := b_HHP_ENABLE AND b_HHP_AZ AND NOT b_limit_unlock AND axisdata[1].Axis_InAb AND axisdata[2].Axis_InAb); // R_TRIG
az1_enable S= R_TRIG_21.Q;
az2_enable S= R_TRIG_21.Q;

// NETWORK 54
TON_2(IN := (az1_enable OR dance_enable_az1) AND NOT b_limit_unlock AND NOT axisdata[1].Axis_Error AND NOT axisdata[2].Axis_Error, PT := t#100ms); // TON
MC_Power_3(Enable := TON_2.Q, Axis := Drive1); // MC_Power

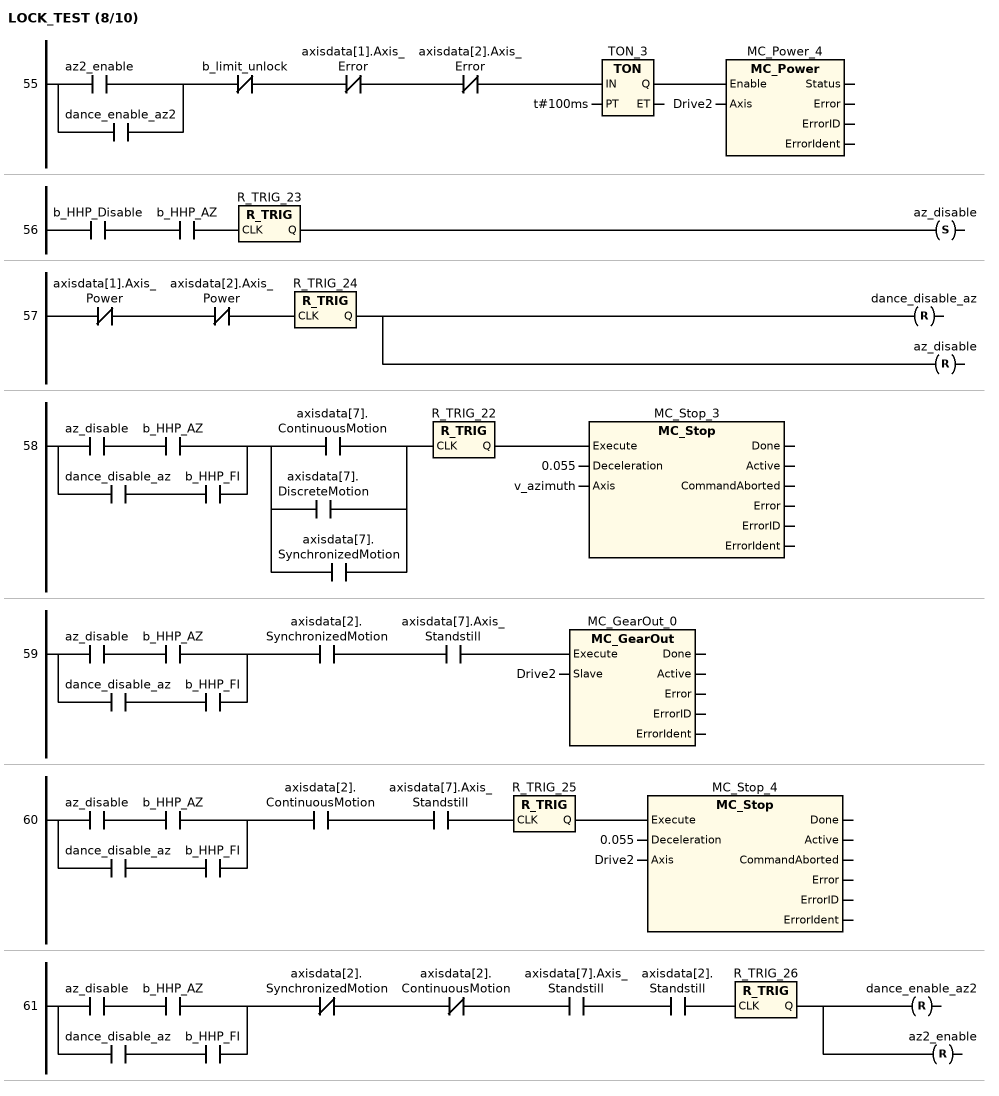
// NETWORK 55
TON_3(IN := (az2_enable OR dance_enable_az2) AND NOT b_limit_unlock AND NOT axisdata[1].Axis_Error AND NOT axisdata[2].Axis_Error, PT := t#100ms); // TON
MC_Power_4(Enable := TON_3.Q, Axis := Drive2); // MC_Power

// NETWORK 56
R_TRIG_23(CLK := b_HHP_Disable AND b_HHP_AZ); // R_TRIG
az_disable S= R_TRIG_23.Q;

// NETWORK 57
R_TRIG_24(CLK := NOT axisdata[1].Axis_Power AND NOT axisdata[2].Axis_Power); // R_TRIG
dance_disable_az R= R_TRIG_24.Q;
az_disable R= R_TRIG_24.Q;

// NETWORK 58
R_TRIG_22(CLK := (az_disable AND b_HHP_AZ OR dance_disable_az AND b_HHP_FI) AND (axisdata[7].ContinuousMotion OR axisdata[7].DiscreteMotion OR axisdata[7].SynchronizedMotion)); // R_TRIG
MC_Stop_3(Execute := R_TRIG_22.Q, Deceleration := 0.055, Axis := v_azimuth); // MC_Stop

// NETWORK 59
MC_GearOut_0(Execute := (az_disable AND b_HHP_AZ OR dance_disable_az AND b_HHP_FI) AND axisdata[2].SynchronizedMotion AND axisdata[7].Axis_Standstill, Slave := Drive2); // MC_GearOut

// NETWORK 60
R_TRIG_25(CLK := (az_disable AND b_HHP_AZ OR dance_disable_az AND b_HHP_FI) AND axisdata[2].ContinuousMotion AND axisdata[7].Axis_Standstill); // R_TRIG
MC_Stop_4(Execute := R_TRIG_25.Q, Deceleration := 0.055, Axis := Drive2); // MC_Stop

// NETWORK 61
R_TRIG_26(CLK := (az_disable AND b_HHP_AZ OR dance_disable_az AND b_HHP_FI) AND NOT axisdata[2].SynchronizedMotion AND NOT axisdata[2].ContinuousMotion AND axisdata[7].Axis_Standstill AND axisdata[2].Standstill); // R_TRIG
dance_enable_az2 R= R_TRIG_26.Q;
az2_enable R= R_TRIG_26.Q;

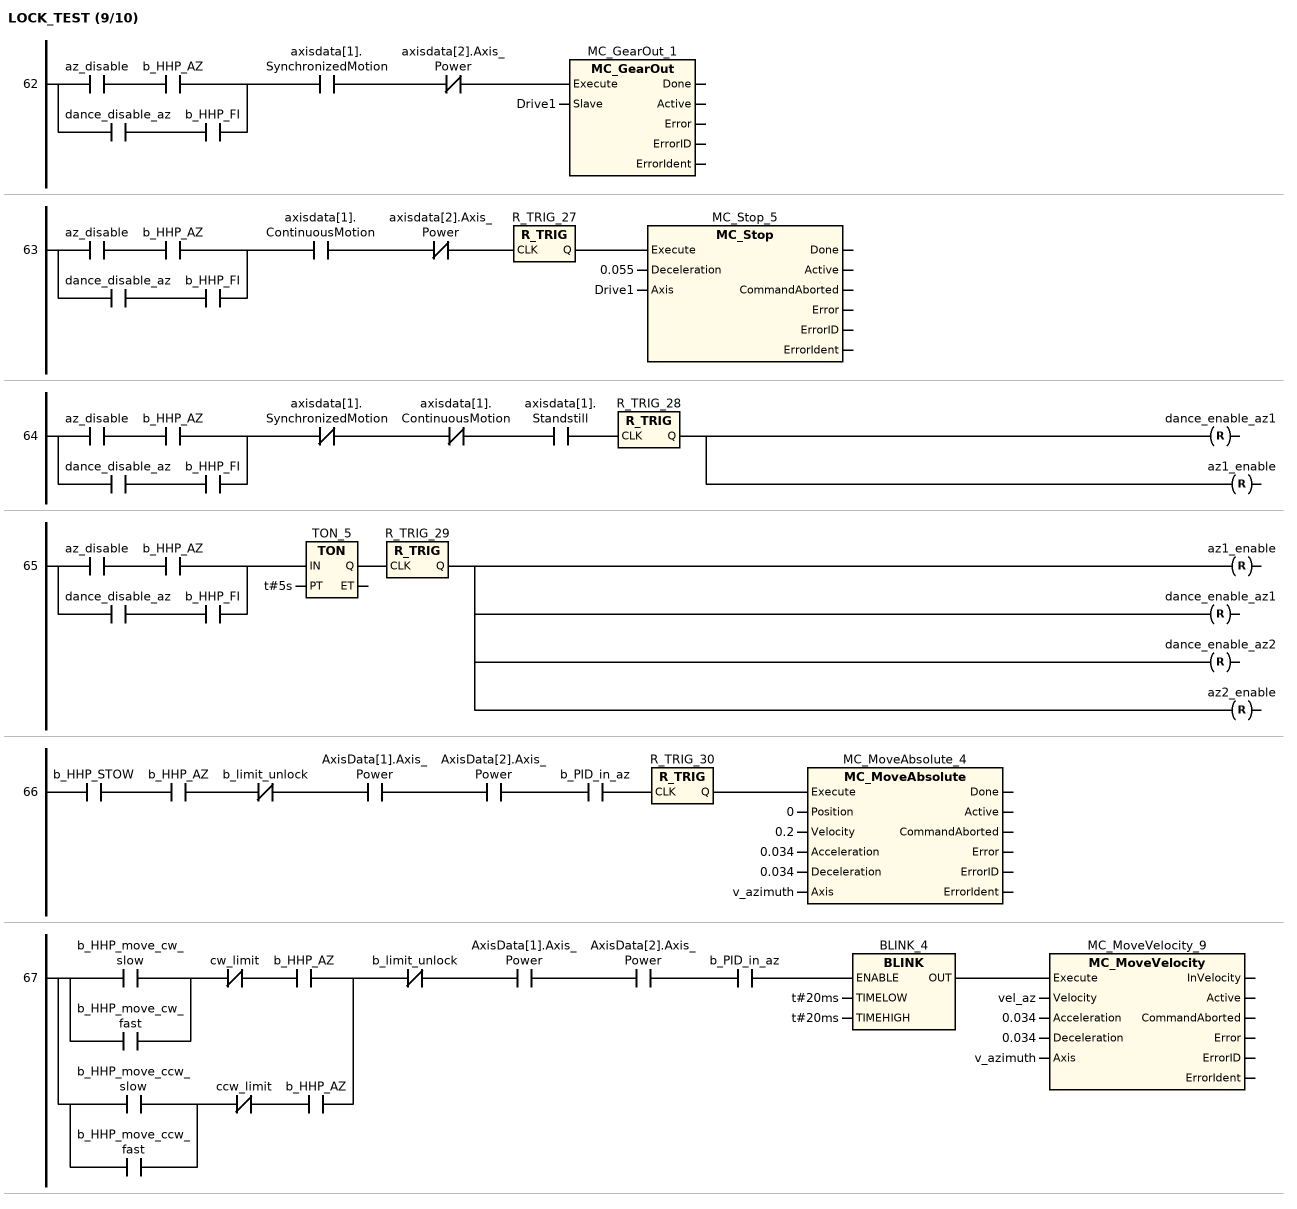
// NETWORK 62
MC_GearOut_1(Execute := (az_disable AND b_HHP_AZ OR dance_disable_az AND b_HHP_FI) AND axisdata[1].SynchronizedMotion AND NOT axisdata[2].Axis_Power, Slave := Drive1); // MC_GearOut

// NETWORK 63
R_TRIG_27(CLK := (az_disable AND b_HHP_AZ OR dance_disable_az AND b_HHP_FI) AND axisdata[1].ContinuousMotion AND NOT axisdata[2].Axis_Power); // R_TRIG
MC_Stop_5(Execute := R_TRIG_27.Q, Deceleration := 0.055, Axis := Drive1); // MC_Stop

// NETWORK 64
R_TRIG_28(CLK := (az_disable AND b_HHP_AZ OR dance_disable_az AND b_HHP_FI) AND NOT axisdata[1].SynchronizedMotion AND NOT axisdata[1].ContinuousMotion AND axisdata[1].Standstill); // R_TRIG
dance_enable_az1 R= R_TRIG_28.Q;
az1_enable R= R_TRIG_28.Q;

// NETWORK 65
TON_5(IN := az_disable AND b_HHP_AZ OR dance_disable_az AND b_HHP_FI, PT := t#5s); // TON
R_TRIG_29(CLK := TON_5.Q); // R_TRIG
az1_enable R= R_TRIG_29.Q;
dance_enable_az1 R= R_TRIG_29.Q;
dance_enable_az2 R= R_TRIG_29.Q;
az2_enable R= R_TRIG_29.Q;

// NETWORK 66
R_TRIG_30(CLK := b_HHP_STOW AND b_HHP_AZ AND NOT b_limit_unlock AND AxisData[1].Axis_Power AND AxisData[2].Axis_Power AND b_PID_in_az); // R_TRIG
MC_MoveAbsolute_4(
    Execute := R_TRIG_30.Q,
    Position := 0,
    Velocity := 0.2,
    Acceleration := 0.034,
    Deceleration := 0.034,
    Axis := v_azimuth); // MC_MoveAbsolute

// NETWORK 67
BLINK_4(
    ENABLE := ((b_HHP_move_cw_slow OR b_HHP_move_cw_fast) AND NOT cw_limit AND b_HHP_AZ OR (b_HHP_move_ccw_slow OR b_HHP_move_ccw_fast) AND NOT ccw_limit AND b_HHP_AZ) AND NOT b_limit_unlock AND AxisData[1].Axis_Power AND AxisData[2].Axis_Power AND b_PID_in_az,
    TIMELOW := t#20ms,
    TIMEHIGH := t#20ms); // BLINK
MC_MoveVelocity_9(
    Execute := BLINK_4.OUT,
    Velocity := vel_az,
    Acceleration := 0.034,
    Deceleration := 0.034,
    Axis := v_azimuth); // MC_MoveVelocity

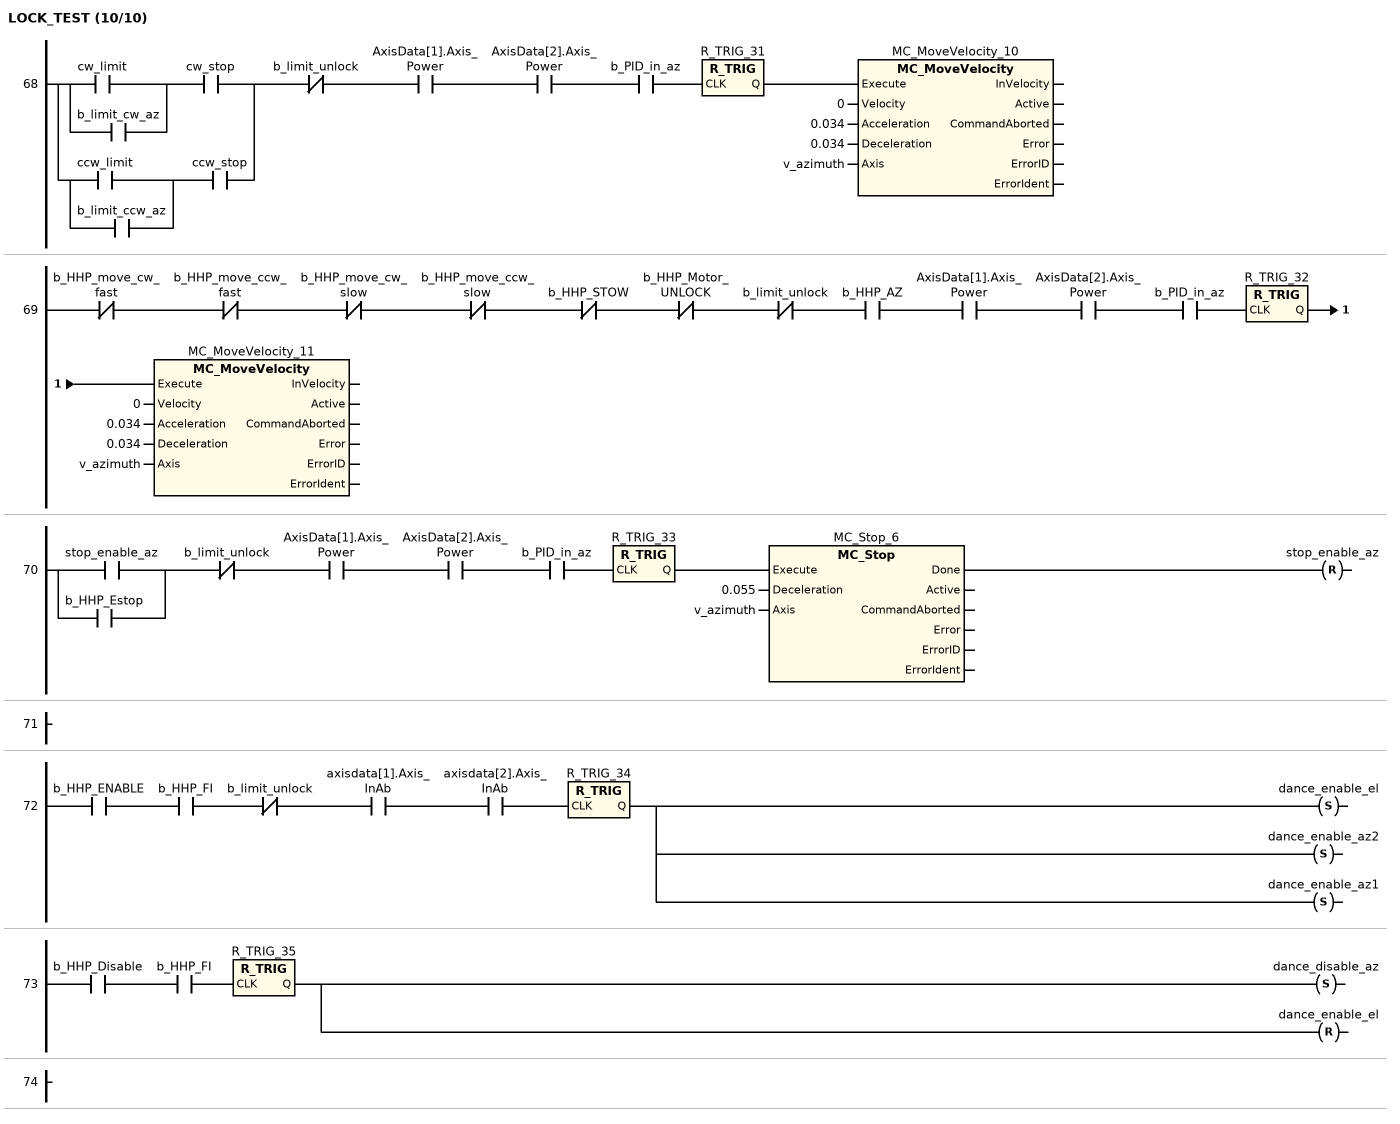
// NETWORK 68
R_TRIG_31(CLK := ((cw_limit OR b_limit_cw_az) AND cw_stop OR (ccw_limit OR b_limit_ccw_az) AND ccw_stop) AND NOT b_limit_unlock AND AxisData[1].Axis_Power AND AxisData[2].Axis_Power AND b_PID_in_az); // R_TRIG
MC_MoveVelocity_10(
    Execute := R_TRIG_31.Q,
    Velocity := 0,
    Acceleration := 0.034,
    Deceleration := 0.034,
    Axis := v_azimuth); // MC_MoveVelocity

// NETWORK 69
R_TRIG_32(CLK := NOT b_HHP_move_cw_fast AND NOT b_HHP_move_ccw_fast AND NOT b_HHP_move_cw_slow AND NOT b_HHP_move_ccw_slow AND NOT b_HHP_STOW AND NOT b_HHP_Motor_UNLOCK AND NOT b_limit_unlock AND b_HHP_AZ AND AxisData[1].Axis_Power AND AxisData[2].Axis_Power AND b_PID_in_az); // R_TRIG
MC_MoveVelocity_11(
    Execute := R_TRIG_32.Q,
    Velocity := 0,
    Acceleration := 0.034,
    Deceleration := 0.034,
    Axis := v_azimuth); // MC_MoveVelocity

// NETWORK 70
R_TRIG_33(CLK := (stop_enable_az OR b_HHP_Estop) AND NOT b_limit_unlock AND AxisData[1].Axis_Power AND AxisData[2].Axis_Power AND b_PID_in_az); // R_TRIG
MC_Stop_6(Execute := R_TRIG_33.Q, Deceleration := 0.055, Axis := v_azimuth); // MC_Stop
stop_enable_az R= MC_Stop_6.Done;

// NETWORK 71

// NETWORK 72
R_TRIG_34(CLK := b_HHP_ENABLE AND b_HHP_FI AND NOT b_limit_unlock AND axisdata[1].Axis_InAb AND axisdata[2].Axis_InAb); // R_TRIG
dance_enable_el S= R_TRIG_34.Q;
dance_enable_az2 S= R_TRIG_34.Q;
dance_enable_az1 S= R_TRIG_34.Q;

// NETWORK 73
R_TRIG_35(CLK := b_HHP_Disable AND b_HHP_FI); // R_TRIG
dance_disable_az S= R_TRIG_35.Q;
dance_enable_el R= R_TRIG_35.Q;

// NETWORK 74

END_PROGRAM

// IndraMotionMlc1/Application/POUs/TCP/P_DRIVE_Modeswitch
(*the program is built for Drive Mode Switch*)
PROGRAM P_DRIVE_Modeswitch
VAR
	dw_drive1_mode: DWORD;
	dw_drive2_mode: DWORD;
	drive1_modeswitch_enable: BOOL;
	drive2_modeswitch_enable: BOOL;

	MB_ReadParameter_0: MB_ReadParameter;
	MB_WriteParameter_0: MB_WriteParameter;
	MB_WriteParameter_1: MB_WriteParameter;
	MB_WriteParameter_2: MB_WriteParameter;
	MB_WriteParameter_3: MB_WriteParameter;
	MB_WriteParameter_4: MB_WriteParameter;
		
	R_TRIG_0: R_TRIG;
	drive1_enable1: BOOL;
	drive1_enable2: BOOL;
	drive1_enable3: BOOL;
	drive1_enable4: BOOL;
	drive1_enable5: BOOL;
	TON_0: TON;
	TON_1: TON;
	TON_2: TON;
	TON_3: TON;
	TON_4: TON;	
	
	MB_ReadParameter_1: MB_ReadParameter;
	MB_WriteParameter_5: MB_WriteParameter;
	MB_WriteParameter_6: MB_WriteParameter;
	MB_WriteParameter_7: MB_WriteParameter;
	MB_WriteParameter_8: MB_WriteParameter;
	MB_WriteParameter_9: MB_WriteParameter;
	
	R_TRIG_1: R_TRIG;
	drive2_enable1: BOOL;
	drive2_enable2: BOOL;
	drive2_enable3: BOOL;
	drive2_enable4: BOOL;
	drive2_enable5: BOOL;
	TON_5: TON;
	TON_6: TON;
	TON_7: TON;
	TON_8: TON;
	TON_9: TON;
	
END_VAR

P_DRIVE_Modeswitch.A_DRIVE_Modeswitch();

IF dw_drive1_mode=16#10B THEN
	drive1_modeswitch_enable:=FALSE;
ELSE
	drive1_modeswitch_enable:=TRUE;
END_IF

IF dw_drive2_mode=16#10B THEN
	drive2_modeswitch_enable:=FALSE;
ELSE
	drive2_modeswitch_enable:=TRUE;
END_IF

ACTION A_DRIVE_Modeswitch:
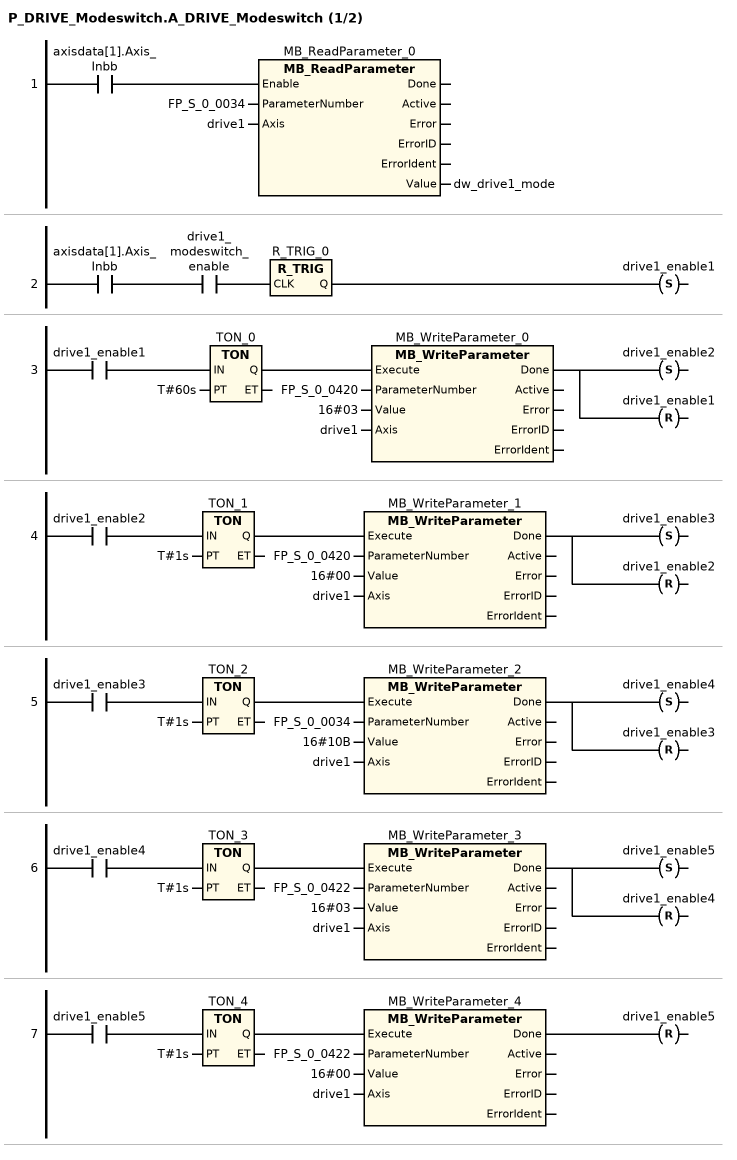
// NETWORK 1
MB_ReadParameter_0(
    Enable := axisdata[1].Axis_Inbb,
    ParameterNumber := FP_S_0_0034,
    Axis := drive1,
    Value => dw_drive1_mode); // MB_ReadParameter

// NETWORK 2
R_TRIG_0(CLK := axisdata[1].Axis_Inbb AND drive1_modeswitch_enable); // R_TRIG
drive1_enable1 S= R_TRIG_0.Q;

// NETWORK 3
TON_0(IN := drive1_enable1, PT := T#60s); // TON
MB_WriteParameter_0(Execute := TON_0.Q, ParameterNumber := FP_S_0_0420, Value := 16#03, Axis := drive1); // MB_WriteParameter
drive1_enable2 S= MB_WriteParameter_0.Done;
drive1_enable1 R= MB_WriteParameter_0.Done;

// NETWORK 4
TON_1(IN := drive1_enable2, PT := T#1s); // TON
MB_WriteParameter_1(Execute := TON_1.Q, ParameterNumber := FP_S_0_0420, Value := 16#00, Axis := drive1); // MB_WriteParameter
drive1_enable3 S= MB_WriteParameter_1.Done;
drive1_enable2 R= MB_WriteParameter_1.Done;

// NETWORK 5
TON_2(IN := drive1_enable3, PT := T#1s); // TON
MB_WriteParameter_2(Execute := TON_2.Q, ParameterNumber := FP_S_0_0034, Value := 16#10B, Axis := drive1); // MB_WriteParameter
drive1_enable4 S= MB_WriteParameter_2.Done;
drive1_enable3 R= MB_WriteParameter_2.Done;

// NETWORK 6
TON_3(IN := drive1_enable4, PT := T#1s); // TON
MB_WriteParameter_3(Execute := TON_3.Q, ParameterNumber := FP_S_0_0422, Value := 16#03, Axis := drive1); // MB_WriteParameter
drive1_enable5 S= MB_WriteParameter_3.Done;
drive1_enable4 R= MB_WriteParameter_3.Done;

// NETWORK 7
TON_4(IN := drive1_enable5, PT := T#1s); // TON
MB_WriteParameter_4(Execute := TON_4.Q, ParameterNumber := FP_S_0_0422, Value := 16#00, Axis := drive1); // MB_WriteParameter
drive1_enable5 R= MB_WriteParameter_4.Done;

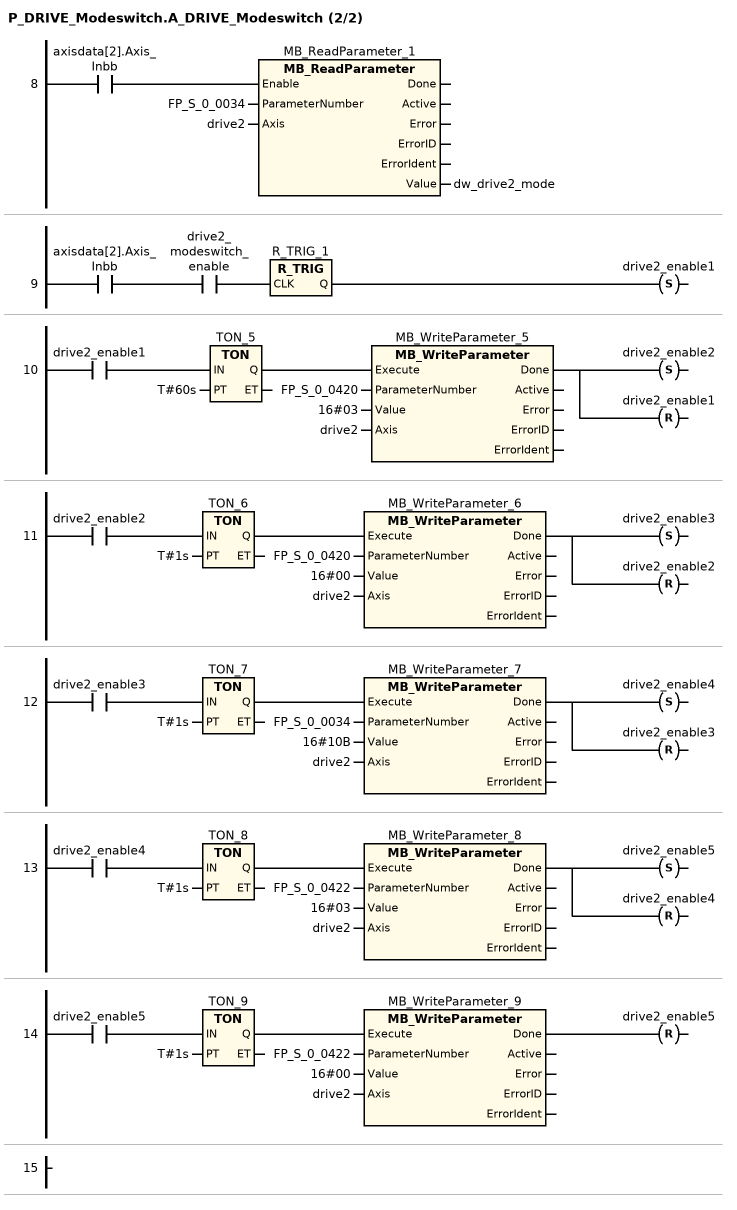
// NETWORK 8
MB_ReadParameter_1(
    Enable := axisdata[2].Axis_Inbb,
    ParameterNumber := FP_S_0_0034,
    Axis := drive2,
    Value => dw_drive2_mode); // MB_ReadParameter

// NETWORK 9
R_TRIG_1(CLK := axisdata[2].Axis_Inbb AND drive2_modeswitch_enable); // R_TRIG
drive2_enable1 S= R_TRIG_1.Q;

// NETWORK 10
TON_5(IN := drive2_enable1, PT := T#60s); // TON
MB_WriteParameter_5(Execute := TON_5.Q, ParameterNumber := FP_S_0_0420, Value := 16#03, Axis := drive2); // MB_WriteParameter
drive2_enable2 S= MB_WriteParameter_5.Done;
drive2_enable1 R= MB_WriteParameter_5.Done;

// NETWORK 11
TON_6(IN := drive2_enable2, PT := T#1s); // TON
MB_WriteParameter_6(Execute := TON_6.Q, ParameterNumber := FP_S_0_0420, Value := 16#00, Axis := drive2); // MB_WriteParameter
drive2_enable3 S= MB_WriteParameter_6.Done;
drive2_enable2 R= MB_WriteParameter_6.Done;

// NETWORK 12
TON_7(IN := drive2_enable3, PT := T#1s); // TON
MB_WriteParameter_7(Execute := TON_7.Q, ParameterNumber := FP_S_0_0034, Value := 16#10B, Axis := drive2); // MB_WriteParameter
drive2_enable4 S= MB_WriteParameter_7.Done;
drive2_enable3 R= MB_WriteParameter_7.Done;

// NETWORK 13
TON_8(IN := drive2_enable4, PT := T#1s); // TON
MB_WriteParameter_8(Execute := TON_8.Q, ParameterNumber := FP_S_0_0422, Value := 16#03, Axis := drive2); // MB_WriteParameter
drive2_enable5 S= MB_WriteParameter_8.Done;
drive2_enable4 R= MB_WriteParameter_8.Done;

// NETWORK 14
TON_9(IN := drive2_enable5, PT := T#1s); // TON
MB_WriteParameter_9(Execute := TON_9.Q, ParameterNumber := FP_S_0_0422, Value := 16#00, Axis := drive2); // MB_WriteParameter
drive2_enable5 R= MB_WriteParameter_9.Done;

// NETWORK 15
END_ACTION

END_PROGRAM

// IndraMotionMlc1/Application/AxisInterface/Visualizations/AxisModes/Axis_Overview
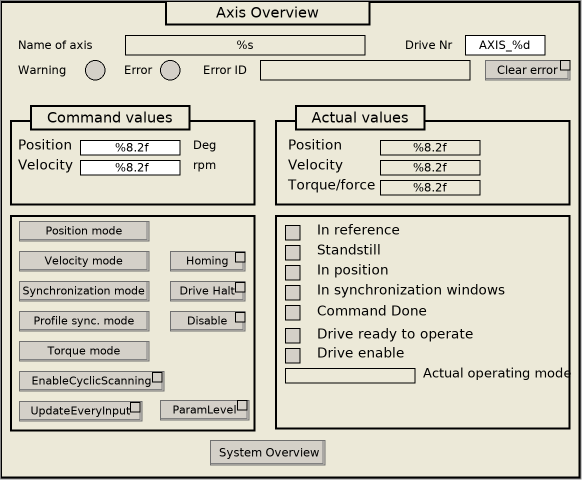
VISUALIZATION Axis_Overview  // 582x480
    Rectangle (0,1 580x477)
    Rectangle (15,35 110x20), "Name of axis"
    Rectangle (385,35 70x20), "Drive Nr"
    Rectangle (125,35 240x20), "%s", text variable: arAxisStatus_gb [VisuAxisNo].Admin.Name
    Ellipse (85,60 20x20), colour toggle: arAxisStatus_gb [VisuAxisNo].Diag.Warning
    Rectangle (15,60 70x20), "Warning"
    Ellipse (160,60 20x20), colour toggle: arAxisStatus_gb [VisuAxisNo].Diag.Error
    Rectangle (115,60 40x20), "Error"
    Rectangle (190,60 60x20), "Error ID"
    Rectangle (260,60 210x20), text list: 'ErrorIDCode', text index: arAxisStatus_gb [VisuAxisNo].Diag.ErrorID
    Button (485,60 85x20), "Clear error"
        tap arAxisCtrl_gb [VisuAxisNo].Admin.ClearError
    Rectangle (560,60 10x10), colour toggle: arAxisCtrl_gb [VisuAxisNo].Admin.ClearError
    Rectangle (165,0 205x25), "Axis Overview"
    Rectangle (10,215 245x216)
    Rectangle (10,120 245x85)
    Rectangle (275,120 295x85)
    Rectangle (295,105 130x25), "Actual values"
    Rectangle (15,135 80x20), "Position"
    Rectangle (285,135 80x20), "Position"
    Rectangle (285,155 80x20), "Velocity"
    Rectangle (285,175 100x20), "Torque/force"
    Rectangle (80,140 100x15), "%8.2f", text variable: arAxisCtrl_gb [VisuAxisNo].PosMode.Position
        OnMouseUp: write arAxisCtrl_gb [VisuAxisNo].PosMode.Position via 
    Rectangle (380,160 100x15), "%8.2f", text variable: AxisData[VisuAxisNo].rActualVelocity_i
    Rectangle (380,180 100x15), "%8.2f", text variable: AxisData[VisuAxisNo].rActualTorqueForce_i
    Rectangle (190,135 40x20), "Deg"
    Rectangle (190,155 40x20), "rpm"
    Rectangle (380,140 100x15), "%8.2f", text variable: AxisData[VisuAxisNo].rActualPosition_i
    Rectangle (80,160 100x15), "%8.2f", text variable: arAxisCtrl_gb [VisuAxisNo].VelMode.Velocity
        OnMouseUp: write arAxisCtrl_gb [VisuAxisNo].VelMode.Velocity via 
    Rectangle (15,155 70x20), "Velocity"
    Button (19,221 130x20), "Position mode"
        OnMouseUp:  Assign=Position_mode, Assign=Position_mode, Type=Assignment
    Button (19,251 130x20), "Velocity mode"
        OnMouseUp:  Assign=Velocity_mode, Assign=Velocity_mode, Type=Assignment
    Button (19,281 130x20), "Synchronization mode"
        OnMouseUp:  Assign=Synchronization_mode, Assign=Synchronization_mode, Type=Assignment
    Button (170,281 75x20), "Drive Halt"
        OnMouseUp: execute { arAxisCtrl_gb [VisuAxisNo].Admin._OpMode.en:=(ModeAh); }
    Rectangle (235,282 10x10), colour toggle: arAxisStatus_gb[VisuAxisNo].Admin._OpModeAck = ModeAH
    Rectangle (30,105 160x25), "Command values"
    Button (170,311 75x20), "Disable"
        OnMouseUp: execute { arAxisCtrl_gb [VisuAxisNo].Admin._OpMode.en:=(ModeAb); }
    Rectangle (235,312 10x10), colour toggle: arAxisStatus_gb[VisuAxisNo].Admin._OpModeAck = ModeAB
    Button (170,251 75x20), "Homing"
        OnMouseUp: execute { arAxisCtrl_gb [VisuAxisNo].Admin._OpMode.en:=(ModeHoming); }
    Rectangle (235,252 10x10), colour toggle: arAxisStatus_gb[VisuAxisNo].Admin._OpModeAck = ModeHoming
    Rectangle (275,215 295x214)
    Rectangle (285,265 15x15), colour toggle: (AxisData[VisuAxisNo].Axis_InPosition) <> 0
    Rectangle (285,285 15x15), colour toggle: (Axisdata[VisuAxisNo].Axis_InSynchron) <> 0
    Rectangle (314,240 100x20), "Standstill"
    Rectangle (314,260 100x20), "In position"
    Rectangle (314,280 250x20), "In synchronization windows"
    Rectangle (285,348 15x15), colour toggle: (AxisData[VisuAxisNo].Axis_Power) <> 0
    Rectangle (285,328 15x15), colour toggle: (AxisData[VisuAxisNo].Axis_InAb) <> 0
    Rectangle (314,343 170x20), "Drive enable"
    Rectangle (314,324 190x20), "Drive ready to operate"
    Rectangle (285,245 15x15), colour toggle: (AxisData[VisuAxisNo].Axis_Standstill) <> 0
    Rectangle (420,363 155x20), "Actual operating mode"
    Rectangle (285,225 15x15), colour toggle: (AxisData[VisuAxisNo].Axis_Homed) <> 0
    Rectangle (314,220 165x20), "In reference"
    Rectangle (285,368 130x15), text list: 'AxisMode', text index: arAxisStatus_gb [VisuAxisNo].Admin._OpModeAck
    Button (210,440 115x25), "System Overview"
        OnMouseUp:  Assign=System_Overview_All_Axis, Type=Assignment
    Rectangle (465,35 80x20), "AXIS_%d", text variable: VisuAxisNo
        OnMouseUp: write VisuAxisNo via 
    Button (19,311 130x20), "Profile sync. mode"
        OnMouseUp:  Assign=Profile_mode, Type=Assignment
    Button (160,400 89x20), "ParamLevel"
        toggle arAxisCtrl_gb[VisuAxisNo].Admin.ParamLevel
    Rectangle (237,400 10x10), colour toggle: arAxisStatus_gb[VisuAxisNo].Admin.ParamLevelAck = TRUE
    Button (19,371 145x20), "EnableCyclicScanning"
        toggle arAxisCtrl_gb[VisuAxisNo].Admin.EnableCyclicScanning
    Rectangle (152,372 10x10), colour toggle: arAxisCtrl_gb[VisuAxisNo].Admin.EnableCyclicScanning
    Button (19,401 123x20), "UpdateEveryInput"
        toggle arAxisCtrl_gb[VisuAxisNo].Admin.UpdateEveryInput
    Rectangle (130,402 10x10), colour toggle: arAxisCtrl_gb[VisuAxisNo].Admin.UpdateEveryInput
    Rectangle (285,305 15x15), colour toggle: (arAxisStatus_gb[VisuAxisNo].Admin.CmdDone) <> 0
    Rectangle (314,301 122x20), "Command Done"
    Button (19,341 130x20), "Torque mode"
        OnMouseUp:  Assign=Torque_mode, Type=Assignment
END_VISUALIZATION

// IndraMotionMlc1/Application/AxisInterface/Visualizations/AxisModes/Position_mode
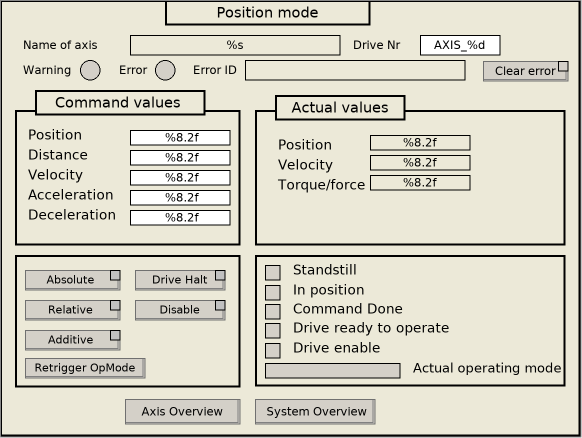
VISUALIZATION Position_mode  // 582x438
    Rectangle (0,0 580x436)
    Rectangle (15,255 225x132)
    Rectangle (165,0 205x25), "Position mode"
    Rectangle (15,110 225x135)
    Rectangle (35,90 170x25), "Command values"
    Rectangle (25,125 80x20), "Position"
    Rectangle (25,145 80x20), "Distance"
    Rectangle (25,165 80x20), "Velocity"
    Rectangle (130,150 100x15), "%8.2f", text variable: arAxisCtrl_gb [VisuAxisNo].PosMode.Distance
        OnMouseUp: write arAxisCtrl_gb [VisuAxisNo].PosMode.Distance via 
    Rectangle (130,170 100x15), "%8.2f", text variable: arAxisCtrl_gb [VisuAxisNo].PosMode.Velocity
        OnMouseUp: write arAxisCtrl_gb [VisuAxisNo].PosMode.Velocity via 
    Rectangle (130,130 100x15), "%8.2f", text variable: arAxisCtrl_gb [VisuAxisNo].PosMode.Position
        OnMouseUp: write arAxisCtrl_gb [VisuAxisNo].PosMode.Position via 
    Rectangle (130,190 100x15), "%8.2f", text variable: arAxisCtrl_gb [VisuAxisNo].PosMode.Acceleration
        OnMouseUp: write arAxisCtrl_gb [VisuAxisNo].PosMode.Acceleration via 
    Rectangle (25,185 100x20), "Acceleration"
    Rectangle (25,205 100x20), "Deceleration"
    Rectangle (130,210 100x15), "%8.2f", text variable: arAxisCtrl_gb [VisuAxisNo].PosMode.Deceleration
        OnMouseUp: write arAxisCtrl_gb [VisuAxisNo].PosMode.Deceleration via 
    Rectangle (255,110 310x135)
    Rectangle (275,95 130x25), "Actual values"
    Rectangle (275,135 80x20), "Position"
    Rectangle (275,155 80x20), "Velocity"
    Rectangle (275,175 100x20), "Torque/force"
    Rectangle (370,155 100x15), "%8.2f", text variable: AxisData[VisuAxisNo].rActualVelocity_i
    Rectangle (370,175 100x15), "%8.2f", text variable: AxisData[VisuAxisNo].rActualTorqueForce_i
    Rectangle (370,135 100x15), "%8.2f", text variable: AxisData[VisuAxisNo].rActualPosition_i
    Button (125,399 115x25), "Axis Overview"
        OnMouseUp:  Assign=Axis_Overview, Assign=Axis_Overview, Type=Assignment
    Rectangle (255,255 310x131)
    Rectangle (265,285 15x15), colour toggle: (AxisData[VisuAxisNo].Axis_InPosition) <> 0
    Rectangle (290,260 100x20), "Standstill"
    Rectangle (290,280 100x20), "In position"
    Rectangle (265,343 15x15), colour toggle: (AxisData[VisuAxisNo].Axis_Power) <> 0
    Rectangle (265,323 15x15), colour toggle: (AxisData[VisuAxisNo].Axis_InAb) <> 0
    Rectangle (290,338 170x20), "Drive enable"
    Rectangle (290,318 190x20), "Drive ready to operate"
    Rectangle (265,265 15x15), colour toggle: (AxisData[VisuAxisNo].Axis_Standstill) <> 0
    Button (25,270 95x20), "Absolute"
        OnMouseUp: execute { arAxisCtrl_gb [VisuAxisNo].Admin._OpMode.en:=(ModePosAbs); }
    Button (25,300 95x20), "Relative"
        OnMouseUp: execute { arAxisCtrl_gb [VisuAxisNo].Admin._OpMode.en:=(ModePosRel); }
    Rectangle (110,270 10x10), colour toggle: (arAxisStatus_gb[VisuAxisNo].Admin.MODE_POS_ABS) <> 0
    Rectangle (110,300 10x10), colour toggle: (arAxisStatus_gb[VisuAxisNo].Admin.MODE_POS_REL) <> 0
    Button (25,330 95x20), "Additive"
        OnMouseUp: execute { arAxisCtrl_gb [VisuAxisNo].Admin._OpMode.en:=(ModePosAdd); }
    Rectangle (110,330 10x10), colour toggle: (arAxisStatus_gb[VisuAxisNo].Admin.MODE_POS_ADD) <> 0
    Button (135,270 90x20), "Drive Halt"
        OnMouseUp: execute { arAxisCtrl_gb [VisuAxisNo].Admin._OpMode.en:=(ModeAh); }
    Rectangle (215,270 10x10), colour toggle: (arAxisStatus_gb[VisuAxisNo].Admin.MODE_AH) <> 0
    Button (135,300 90x20), "Disable"
        OnMouseUp: execute { arAxisCtrl_gb [VisuAxisNo].Admin._OpMode.en:=(ModeAb); }
    Rectangle (215,300 10x10), colour toggle: (arAxisStatus_gb[VisuAxisNo].Admin._OpModeAck = ModeAb) <> 0
    Rectangle (265,363 135x15), text list: 'AxisMode', text index: arAxisStatus_gb [VisuAxisNo].Admin._OpModeAck
    Rectangle (410,358 155x20), "Actual operating mode"
    Rectangle (20,35 110x20), "Name of axis"
    Rectangle (350,35 70x20), "Drive Nr"
    Rectangle (130,35 210x20), "%s", text variable: arAxisStatus_gb [VisuAxisNo].Admin.Name
    Ellipse (80,60 20x20), colour toggle: arAxisStatus_gb [VisuAxisNo].Diag.Warning
    Rectangle (20,60 70x20), "Warning"
    Ellipse (155,60 20x20), colour toggle: arAxisStatus_gb [VisuAxisNo].Diag.Error
    Rectangle (110,60 40x20), "Error"
    Rectangle (180,60 60x20), "Error ID"
    Rectangle (245,60 220x20), text list: 'ErrorIDCode', text index: arAxisStatus_gb [VisuAxisNo].Diag.ErrorID
    Button (255,399 120x25), "System Overview"
        OnMouseUp:  Assign=System_Overview_All_Axis, Assign=System_Overview_All_Axis, Type=Assignment
    Rectangle (420,35 80x20), "AXIS_%d", text variable: VisuAxisNo
        OnMouseUp: write VisuAxisNo via 
    Button (483,61 85x20), "Clear error"
        tap arAxisCtrl_gb [VisuAxisNo].Admin.ClearError
    Rectangle (558,61 10x10), colour toggle: arAxisCtrl_gb [VisuAxisNo].Admin.ClearError
    Button (25,358 120x20), "Retrigger OpMode"
        tap arAxisCtrl_gb[VisuAxisNo].Admin.RetriggerOpMode
    Rectangle (265,304 15x15), colour toggle: (arAxisStatus_gb[VisuAxisNo].Admin.CmdDone) <> 0
    Rectangle (290,299 122x20), "Command Done"
END_VISUALIZATION

// IndraMotionMlc1/Application/AxisInterface/Visualizations/AxisModes/Profile_mode
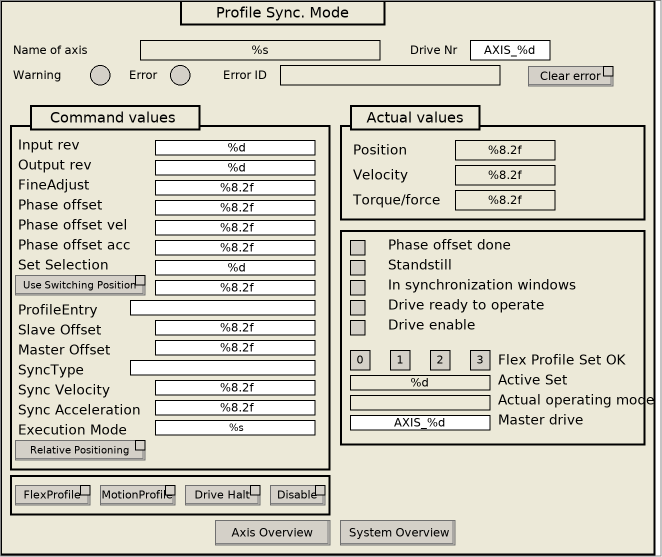
VISUALIZATION Profile_mode  // 662x557
    Rectangle (0,0 655x555)
    Rectangle (340,230 305x215)
    Rectangle (10,475 320x40)
    Button (100,485 75x20), "MotionProfile"
        OnMouseUp: execute { arAxisCtrl_gb [VisuAxisNo].Admin._OpMode.en:=(ModeSyncProfile); }
    Rectangle (180,0 205x25), "Profile Sync. Mode"
    Rectangle (10,125 320x345)
    Rectangle (30,105 170x25), "Command values"
    Rectangle (15,135 120x20), "Input rev"
    Rectangle (15,155 120x20), "Output rev"
    Rectangle (15,175 120x20), "FineAdjust"
    Rectangle (155,160 160x15), "%d", text variable: arAxisCtrl_gb [VisuAxisNo].SyncMode.OutputRevolution
        OnMouseUp: write arAxisCtrl_gb [VisuAxisNo].SyncMode.OutputRevolution via 
    Rectangle (155,180 160x15), "%8.2f", text variable: arAxisCtrl_gb [VisuAxisNo].SyncMode.FineAdjust
        OnMouseUp: write arAxisCtrl_gb [VisuAxisNo].SyncMode.FineAdjust via 
    Rectangle (155,140 160x15), "%d", text variable: arAxisCtrl_gb [VisuAxisNo].SyncMode.InputRevolution
        OnMouseUp: write arAxisCtrl_gb [VisuAxisNo].SyncMode.InputRevolution via 
    Rectangle (15,195 120x20), "Phase offset"
    Rectangle (155,200 160x15), "%8.2f", text variable: arAxisCtrl_gb [VisuAxisNo].SyncMode.PhaseOffset
        OnMouseUp: write arAxisCtrl_gb [VisuAxisNo].SyncMode.PhaseOffset via 
    Rectangle (155,220 160x15), "%8.2f", text variable: arAxisCtrl_gb [VisuAxisNo].SyncMode.PhaseOffsetVel
        OnMouseUp: write arAxisCtrl_gb [VisuAxisNo].SyncMode.PhaseOffsetVel via 
    Rectangle (15,215 140x20), "Phase offset vel"
    Rectangle (15,235 140x20), "Phase offset acc"
    Rectangle (155,240 160x15), "%8.2f", text variable: arAxisCtrl_gb [VisuAxisNo].SyncMode.PhaseOffsetAcc
        OnMouseUp: write arAxisCtrl_gb [VisuAxisNo].SyncMode.PhaseOffsetAcc via 
    Rectangle (340,125 305x95)
    Rectangle (350,105 130x25), "Actual values"
    Rectangle (350,140 100x20), "Position"
    Rectangle (350,165 100x20), "Velocity"
    Rectangle (350,190 110x20), "Torque/force"
    Rectangle (455,165 100x20), "%8.2f", text variable: AxisData[VisuAxisNo].rActualVelocity_i
    Rectangle (455,190 100x20), "%8.2f", text variable: AxisData[VisuAxisNo].rActualTorqueForce_i
    Rectangle (455,140 100x20), "%8.2f", text variable: AxisData[VisuAxisNo].rActualPosition_i
    Button (15,485 75x20), "FlexProfile"
        OnMouseUp: execute { arAxisCtrl_gb [VisuAxisNo].Admin._OpMode.en:=(ModeFlexProfile); }
    Rectangle (80,485 10x10), colour toggle: (arAxisStatus_gb[VisuAxisNo].Admin.MODE_FLEX_PROFILE) <> 0
    Rectangle (350,280 15x15), colour toggle: (AxisData[VisuAxisNo].Axis_InSynchron) <> 0
    Rectangle (385,255 100x20), "Standstill"
    Rectangle (385,275 240x20), "In synchronization windows"
    Rectangle (350,320 15x15), colour toggle: (AxisData[VisuAxisNo].Axis_Power) <> 0
    Rectangle (350,300 15x15), colour toggle: (AxisData[VisuAxisNo].Axis_InAb) <> 0
    Rectangle (385,295 190x20), "Drive ready to operate"
    Rectangle (350,260 15x15), colour toggle: (AxisData[VisuAxisNo].Axis_Standstill) <> 0
    Button (185,485 75x20), "Drive Halt"
        OnMouseUp: execute { arAxisCtrl_gb [VisuAxisNo].Admin._OpMode.en:=(ModeAh); }
    Rectangle (250,485 10x10), colour toggle: (arAxisStatus_gb[VisuAxisNo].Admin.MODE_AH) <> 0
    Button (270,485 55x20), "Disable"
        OnMouseUp: execute { arAxisCtrl_gb [VisuAxisNo].Admin._OpMode.en:=(ModeAb); }
    Rectangle (315,485 10x10), colour toggle: (arAxisStatus_gb[VisuAxisNo].Admin._OpModeAck = ModeAb) <> 0
    Rectangle (350,240 15x15), colour toggle: arAxisStatus_gb [VisuAxisNo].SyncMode.PhasingSlaveDone
    Rectangle (385,235 250x20), "Phase offset done"
    Rectangle (10,40 120x20), "Name of axis"
    Rectangle (390,40 70x20), "Drive Nr"
    Rectangle (140,40 240x20), "%s", text variable: arAxisStatus_gb [VisuAxisNo].Admin.Name
    Ellipse (90,65 20x20), colour toggle: arAxisStatus_gb [VisuAxisNo].Diag.Warning
    Rectangle (10,65 70x20), "Warning"
    Ellipse (170,65 20x20), colour toggle: arAxisStatus_gb [VisuAxisNo].Diag.Error
    Rectangle (120,65 40x20), "Error"
    Rectangle (200,65 70x20), "Error ID"
    Rectangle (280,65 220x20), text list: 'ErrorIDCode', text index: arAxisStatus_gb [VisuAxisNo].Diag.ErrorID
    Button (215,520 115x25), "Axis Overview"
        OnMouseUp:  Assign=Axis_Overview, Assign=Axis_Overview, Type=Assignment
    Button (340,520 115x25), "System Overview"
        OnMouseUp:  Assign=System_Overview_All_Axis, Assign=System_Overview_All_Axis, Type=Assignment
    Rectangle (385,315 170x20), "Drive enable"
    Rectangle (470,40 80x20), "AXIS_%d", text variable: VisuAxisNo
        OnMouseUp: write VisuAxisNo via 
    Rectangle (350,415 140x15), "AXIS_%d", text variable: arAxisCtrl_gb [VisuAxisNo].SyncMode.Master.AxisNo
        OnMouseUp: write arAxisCtrl_gb [VisuAxisNo].SyncMode.Master.AxisNo via 
    Rectangle (495,410 100x20), "Master drive"
    Rectangle (350,395 140x15), text list: 'AxisMode', text index: arAxisStatus_gb [VisuAxisNo].Admin._OpModeAck
    Rectangle (495,390 165x20), "Actual operating mode"
    Rectangle (15,255 140x20), "Set Selection"
    Rectangle (155,260 160x15), "%d", text variable: arAxisCtrl_gb [VisuAxisNo].SyncMode.Profile.SetSelection
        OnMouseUp: write arAxisCtrl_gb [VisuAxisNo].SyncMode.Profile.SetSelection via 
    Button (15,440 130x20), "Relative Positioning"
        toggle arAxisCtrl_gb [VisuAxisNo].SyncMode.Profile.RelativePositioning
    Rectangle (165,485 10x10), colour toggle: (arAxisStatus_gb[VisuAxisNo].Admin.MODE_SYNC_PROFILE) <> 0
    Rectangle (135,440 10x10), colour toggle: (arAxisCtrl_gb[VisuAxisNo].SyncMode.Profile.RelativePositioning) <> 0
    Button (15,275 130x20), "Use Switching Position"
        toggle arAxisCtrl_gb [VisuAxisNo].SyncMode.Profile.UseSwitchingPosition
    Rectangle (155,280 160x15), "%8.2f", text variable: arAxisCtrl_gb [VisuAxisNo].SyncMode.Profile.SwitchingPosition
        OnMouseUp: write arAxisCtrl_gb [VisuAxisNo].SyncMode.Profile.SwitchingPosition via 
    Rectangle (130,300 185x15), text list: 'ProfileEntry', text index: arAxisCtrl_gb [VisuAxisNo].SyncMode.Profile.ProfileEntry
        OnMouseUp: write arAxisCtrl_gb [VisuAxisNo].SyncMode.Profile.ProfileEntry via 
    Rectangle (155,320 160x15), "%8.2f", text variable: arAxisCtrl_gb [VisuAxisNo].SyncMode.Profile.SlaveOffset
        OnMouseUp: write arAxisCtrl_gb [VisuAxisNo].SyncMode.Profile.SlaveOffset via 
    Rectangle (155,340 160x15), "%8.2f", text variable: arAxisCtrl_gb [VisuAxisNo].SyncMode.Profile.MasterOffset
        OnMouseUp: write arAxisCtrl_gb [VisuAxisNo].SyncMode.Profile.MasterOffset via 
    Rectangle (15,300 140x20), "ProfileEntry"
    Rectangle (15,320 140x20), "Slave Offset"
    Rectangle (15,340 140x20), "Master Offset"
    Rectangle (130,360 185x15), text list: 'SyncType', text index: arAxisCtrl_gb [VisuAxisNo].SyncMode.Profile.SyncType
        OnMouseUp: write arAxisCtrl_gb [VisuAxisNo].SyncMode.Profile.SyncType via 
    Rectangle (155,380 160x15), "%8.2f", text variable: arAxisCtrl_gb [VisuAxisNo].SyncMode.SyncVelocity
        OnMouseUp: write arAxisCtrl_gb [VisuAxisNo].SyncMode.SyncVelocity via Edit
    Rectangle (155,400 160x15), "%8.2f", text variable: arAxisCtrl_gb [VisuAxisNo].SyncMode.SyncAcceleration
        OnMouseUp: write arAxisCtrl_gb [VisuAxisNo].SyncMode.SyncAcceleration via Edit
    Rectangle (155,420 160x15), "%s", text list: 'ExecutionMode', text index: arAxisCtrl_gb [VisuAxisNo].SyncMode.Profile.ExecutionMode
        OnMouseUp: write arAxisCtrl_gb [VisuAxisNo].SyncMode.Profile.ExecutionMode via 
    Rectangle (15,360 140x20), "SyncType"
    Rectangle (15,380 140x20), "Sync Velocity"
    Rectangle (15,400 140x20), "Sync Acceleration"
    Rectangle (15,420 140x20), "Execution Mode"
    Rectangle (135,275 10x10), colour toggle: (arAxisCtrl_gb[VisuAxisNo].SyncMode.Profile.UseSwitchingPosition) <> 0
    Rectangle (350,375 140x15), "%d", text variable: arAxisStatus_gb [VisuAxisNo].SyncMode.ProfileActiveSet
    Rectangle (495,370 165x20), "Active Set"
    Rectangle (350,350 20x20), "0", colour toggle: (AxisData[VisuAxisNo].FlexProfil_Set0_Ok) <> 0
    Rectangle (390,350 20x20), "1", colour toggle: (AxisData[VisuAxisNo].FlexProfil_Set1_Ok) <> 0
    Rectangle (430,350 20x20), "2", colour toggle: (AxisData[VisuAxisNo].FlexProfil_Set2_Ok) <> 0
    Rectangle (470,350 20x20), "3", colour toggle: (AxisData[VisuAxisNo].FlexProfil_Set3_Ok) <> 0
    Rectangle (495,350 130x20), "Flex Profile Set OK"
    Button (528,66 85x20), "Clear error"
        tap arAxisCtrl_gb [VisuAxisNo].Admin.ClearError
    Rectangle (603,66 10x10), colour toggle: arAxisCtrl_gb [VisuAxisNo].Admin.ClearError
END_VISUALIZATION

// IndraMotionMlc1/Application/AxisInterface/Visualizations/AxisModes/Synchronization_mode
